// TwinCAT 3 PLC project IDPLC
// ProgramVersion: 3.1.4024.12
// libraries:
//   Tc2_Drive, * (Beckhoff Automation GmbH)
//   Tc2_EtherCAT, * (Beckhoff Automation GmbH)
//   Tc2_Math, * (Beckhoff Automation GmbH)
//   Tc2_MC2, * (Beckhoff Automation GmbH)
//   Tc2_NC, * (Beckhoff Automation GmbH)
//   Tc2_NcDrive, * (Beckhoff Automation GmbH)
//   Tc2_SerialCom, * (Beckhoff Automation GmbH)
//   Tc2_Standard, * (Beckhoff Automation GmbH)
//   Tc2_System, * (Beckhoff Automation GmbH)
//   Tc2_Utilities, * (Beckhoff Automation GmbH)
//   Tc3_Module, * (Beckhoff Automation GmbH)
// project tree:
//   DUTs/ DUT.TcDUT (not stored), DUT_SENSOR_DATAS_1.TcDUT (not stored), DUT_SENSOR_DATAS_8.TcDUT (not stored), DUT_SENSOR_DATAS_2.TcDUT (not stored), DUT_SENSOR_DATAS_3.TcDUT (not stored), DUT_SENSOR_DATAS_4.TcDUT (not stored), DUT_SENSOR_DATAS_5.TcDUT (not stored), DUT_SENSOR_DATAS_6.TcDUT (not stored), DUT_SENSOR_DATAS_7.TcDUT (not stored), Struct_M_Compensation.TcDUT (not stored), Struct_M_lakeshore.TcDUT (not stored), ST_P180.TcDUT (not stored), ST_P182.TcDUT (not stored), ST_P183.TcDUT (not stored), ST_PolarizationParam.TcDUT
//   GVLs/ Global_Variables.TcGVL, Variable_Configuration.TcGVL (not stored)
//   / PlcTask.TcTTO, RecipeManager.TcRMO (not stored), Task_SAFE.TcTTO
//   POUs/0.UserMode/ F_GetSysTime.TcPOU (not stored), UserMode.TcPOU
//   POUs/1.CarrierMode/GapMode/ BCGapMode.TcPOU, GapMode.TcPOU
//   POUs/1.CarrierMode/SingleCarrierMode/ SingleCarrierMode.TcPOU
//   POUs/2.SingleMotorMode/DebugMode/ DebugMode.TcPOU
//   POUs/2.SingleMotorMode/TaperMode/ TaperMode.TcPOU
//   POUs/CommonFB/ExternFB/ FB_LedShow.TcPOU (not stored), FB_PlcEmergencyStop.TcPOU (not stored)
//   POUs/CommonFB/MainFB/ FB_CoupleAxis.TcPOU (not stored), FB_DecoupleAxis.TcPOU (not stored), FB_Move.TcPOU, FB_Power.TcPOU, FB_SetAxisPosition.TcPOU, FB_SetMotorAxisPosition.TcPOU (not stored), FB_SetPhaseLowerMotorAxisPosition.TcPOU, FB_SetPhaseUpperAxisPosition.TcPOU, FB_SetPhaseLowerAxisPosition.TcPOU, FB_SetPhaseUpperMotorAxisPosition.TcPOU, FB_Stop.TcPOU
//   POUs/ MAIN.TcPOU
//   POUs/MainPRG/ FB_CheckCoupleStatus.TcPOU (not stored)
//   POUs/PolarStatusFB/ FB_PolarizationState.TcPOU
//   POUs/RS232/ BackgroundEL.TcPOU (not stored), FB_SerialCom.TcPOU (not stored)
//   POUs/TiltSensor/ FB_Simple_MovingAvg.TcPOU (not stored), SAFE.TcPOU

CONFIGURATION IDPLC
    RESOURCE PLC ON TwinCAT3
        TASK PlcTask(INTERVAL := T#10ms, PRIORITY := 20);
        TASK Task_SAFE(INTERVAL := T#1ms, PRIORITY := 1);
        PROGRAM MAIN WITH PlcTask : MAIN;
        PROGRAM SAFE WITH Task_SAFE : SAFE;
    END_RESOURCE
END_CONFIGURATION

// ---- DUTs/ST_PolarizationParam.TcDUT
TYPE ST_PolarizationParam:
STRUCT
    // HM 水平偏振
    Upper_HM  : LREAL := 0.0;
    Lower_HM  : LREAL := 0.0;

    // VM 垂直偏振 (两种情况)
    Upper_VM1 : LREAL := 42.8;
    Lower_VM1 : LREAL := -42.8;
    Upper_VM2 : LREAL := -42.8;
    Lower_VM2 : LREAL := 42.8;

    // LC 左旋圆偏振
    Upper_LC  : LREAL := 64.2;
    Lower_LC  : LREAL := -21.4;

    // RC 右旋圆偏振
    Upper_RC  : LREAL := -64.2;
    Lower_RC  : LREAL := 21.4;

    // 容差
    Tolerance : LREAL := 2.0;
END_STRUCT
END_TYPE

// ---- GVLs/Global_Variables.TcGVL
//{attribute 'Tc2GvlVarNames'}
VAR_GLOBAL
(*IDControl Ready*)
	IDControlReady:BOOL;
(*Maintenance Mode*)
	MaintenanceMode:BOOL;
	MaintenanceModeLed:BOOL;
(*RecipeDescription*)
	RecipeSavedDate:STRING;
	RecipeDescription:STRING;
(*key Command*)
	btn_Power:BOOL;
	btn_PowerOn: BOOL;
	btn_PowerOff: BOOL;
(*Reset*)
btn_Reset:BOOL;
(*Error Massage*)
	Error:BOOL;
	ErrorID:DINT;
	ErrorDescription:STRING;
(*加载配方参数*)
	LoadRecipeParameters:BOOL;
	loadParametersDone:BOOL;
(*Max Velocity Global*)
	MaxVelocityGlobalVelocity : LREAL;
(*设置光栅bias done *)	
	PositionBiasDone:BOOL;
(*Drive Status*)
	DriveStatus:DINT;//1:Drive Ready;2:Axis is in operation;0:Others
(*回程差*)
	HysteresisError:LREAL;
	HysteresisError_PhaseUpper:LREAL:=0.1;
	HysteresisError_PhaseLower:LREAL:=0.1;
(*光栅漂移误差阈值*)
	LEDriftErrorThreshold:LREAL:=0.001;
	LEDriftErrorThreshold_PhaseUpper:LREAL:=0.001;
	LEDriftErrorThreshold_PhaseLower:LREAL:=0.001;
(*Lag Distance threshold*)
	PosDiff_LeftTopLin: LREAL:=0.5;
	PosDiff_RightTopLin:LREAL:=0.5;
	PosDiff_LeftBottomLin:LREAL:=0.5;
	PosDiff_RightBottomLin:LREAL:=0.5;
	PosDiff_PhaseUpperLin:LREAL:=0.5;
	PosDiff_PhaseLowerLin:LREAL:=0.5;
(*UserMode Threshold*)
	Threshold_UserTopPos: LREAL:=0.5;
	Threshold_UserBottomPos: LREAL:=0.5;
	Threshold_UserLeftPos: LREAL:=0.5;
	Threshold_UserRightPos: LREAL:=0.5;
	Threshold_UserTopVelo: LREAL:=0.5;
	Threshold_UserBottomVelo: LREAL:=0.5;
	Threshold_UserLeftVelo: LREAL:=0.5;
	Threshold_UserRightVelo: LREAL:=0.5;
	//
	Range_UserTaperPos:LREAL:=4.01;
	Range_UserTaperVelo:LREAL:=1.01;
	//Diff_TaperLeftPos:LREAL:=0.01;
	//Diff_TaperLeftVelo:LREAL:=0.2;
	//Diff_TaperRightPos:LREAL:=0.05;
	//Diff_TaperRightVelo:LREAL:=0.5;
	//Taper_BeyondRangePositive:BOOL;
	//Diff_TaperTopPos:LREAL:=0.05;
	//Diff_TaperBottomPos:LREAL:=0.05;
	//Taper_BeyondRangeNegtive:BOOL;
(*BCGap Threshold*)
	Threshold_BCTopPos: LREAL:=0.5;
	Threshold_BCBottomPos: LREAL:=0.5;
	Threshold_BCLeftPos: LREAL:=0.5;
	Threshold_BCRightPos: LREAL:=0.5;
	Threshold_BCTopVelo: LREAL:=0.5;
	Threshold_BCBottomVelo: LREAL:=0.5;
	Threshold_BCLeftVelo: LREAL:=0.5;
	Threshold_BCRightVelo: LREAL:=0.5;
(*DebugMode Threshold*)
	Threshold_TopPos_Debug: LREAL:=4;
	Threshold_BottomPos_Debug: LREAL:=4;
	Threshold_LeftPos_Debug: LREAL:=4;
	Threshold_RightPos_Debug: LREAL:=4;
	//单轴目标位置和当前位置之差，阈值
	Threshold_LeftTopPos_Debug: LREAL:=0.4;	
	Threshold_RightTopPos_Debug: LREAL:=0.4;
	Threshold_LeftBottomPos_Debug: LREAL:=0.4;
	Threshold_RightBottomPos_Debug: LREAL:=0.4;
(*Taper Mode Threshold*)
	Range_TaperPos:LREAL:=5.01;
	Range_TaperVelo:LREAL:=1.01;
	Threshold_TaperLeftPos:LREAL:=0.01;
	Threshold_TaperLeftVelo:LREAL:=0.2;
	Threshold_TaperRightPos:LREAL:=0.05;
	Threshold_TaperRightVelo:LREAL:=0.5;
	Taper_BeyondRangePositive:BOOL;
	Threshold_TaperTopPos:LREAL:=0.05;
	Threshold_TaperBottomPos:LREAL:=0.05;
	Taper_BeyondRangeNegtive:BOOL;
(*SingleCarrierMode threshold*)
	Threshold_TopPos_SingleCarrier: LREAL:=2;
	Threshold_BottomPos_SingleCarrier: LREAL:=2;
	Threshold_LeftPos_SingleCarrier: LREAL:=2;
	Threshold_RightPos_SingleCarrier: LREAL:=2;
	Threshold_TopVelo_SingleCarrier: LREAL:=2;
	Threshold_BottomVelo_SingleCarrier: LREAL:=2;
	Threshold_LeftVelo_SingleCarrier: LREAL:=2;
	Threshold_RightVelo_SingleCarrier: LREAL:=2;
		(*Moving or notmoving*)
	moveDoneAllAxis: BOOL;
	moveStatusLeftTop: BOOL;
	moveStatusRightTop: BOOL;
	moveStatusLeftBottom: BOOL;
	moveStatusRightBottom: BOOL;
	moveStatusPhaseUpper: BOOL;
	moveStatusPhaseLower: BOOL;
	moveStatusAllAxis: BOOL;
	moveStatusAnyAxis: BOOL;
	
	(*Moving or notmoving-Motor*)
	moveDoneAllAxisMotor: BOOL;
	moveStatusLeftTopMotor: BOOL;
	moveStatusRightTopMotor: BOOL;
	moveStatusLeftBottomMotor: BOOL;
	moveStatusRightBottomMotor: BOOL;
	moveStatusPhaseUpperMotor: BOOL;
	moveStatusPhaseLowerMotor: BOOL;
	moveStatusAllAxisMotor: BOOL;
	moveStatusAnyAxisMotor: BOOL;	
	moveStatusGap:BOOL;
(*Compensation Value*)
	M_Compensation:ARRAY[1..18] OF Struct_M_Compensation
:=[
(Encoder:=0,	LeftTop:=0,	RightTop:=0,		LeftBottom:=0,	RightBottom:=0,	InRange:=FALSE),
(Encoder:=5.5,	LeftTop:=5.5,	RightTop:=5.5,	LeftBottom:=5.5,	RightBottom:=5.5,	InRange:=FALSE),
(Encoder:=6.0,	LeftTop:=6.0,	RightTop:=6.0,	LeftBottom:=6.0,	RightBottom:=6.0,	InRange:=FALSE),
(Encoder:=6.5,	LeftTop:=6.5,	RightTop:=6.5,	LeftBottom:=6.5,	RightBottom:=6.5,	InRange:=FALSE),
(Encoder:=7.5,	LeftTop:=7.5,	RightTop:=7.5,	LeftBottom:=7.5,	RightBottom:=7.5,	InRange:=FALSE),
(Encoder:=8.5,	LeftTop:=8.5,	RightTop:=8.5,	LeftBottom:=8.5,	RightBottom:=8.5,	InRange:=FALSE),
(Encoder:=9.5,	LeftTop:=9.5,	RightTop:=9.5,	LeftBottom:=9.5,	RightBottom:=9.5,	InRange:=FALSE),
(Encoder:=10.5,	LeftTop:=10.5,	RightTop:=10.5,	LeftBottom:=10.5,	RightBottom:=10.5,		InRange:=FALSE),
(Encoder:=11.5,	LeftTop:=11.5,	RightTop:=11.5,	LeftBottom:=11.5,	RightBottom:=11.5,		InRange:=FALSE),
(Encoder:=30.0,	LeftTop:=30.0,	RightTop:=30.0,	LeftBottom:=30.0,	RightBottom:=30.0,		InRange:=FALSE),
(Encoder:=100.0,	LeftTop:=100.0,	RightTop:=100.0,	LeftBottom:=100.0,	RightBottom:=100.0,		InRange:=FALSE),
(Encoder:=110.0,	LeftTop:=110.0,	RightTop:=110.0,	LeftBottom:=110.0,	RightBottom:=110.0,		InRange:=FALSE),
(Encoder:=120.0,	LeftTop:=120.0,	RightTop:=120.0,	LeftBottom:=120.0,	RightBottom:=120.0,		InRange:=FALSE),
(Encoder:=130.0,	LeftTop:=130.0,	RightTop:=130.0,	LeftBottom:=130.0,	RightBottom:=130.0,		InRange:=FALSE),
(Encoder:=140.0,	LeftTop:=140.0,	RightTop:=140.0,	LeftBottom:=140.0,	RightBottom:=140.0,		InRange:=FALSE),
(Encoder:=150.0,	LeftTop:=150.0,	RightTop:=150.0,	LeftBottom:=150.0,	RightBottom:=150.0,		InRange:=FALSE),
(Encoder:=160.0,	LeftTop:=160.0,	RightTop:=160.0,	LeftBottom:=160.0,	RightBottom:=160.0,		InRange:=FALSE),
(Encoder:=3000.001,	LeftTop:=3000.001,	RightTop:=3000.001,		LeftBottom:=3000.001,	RightBottom:=3000.001,	InRange:=FALSE)];

(*simulation OR NOT*)
	simulation:BOOL;
(*USELinearEncoeder*)
	USELinearEncoder:BOOL:=TRUE;
(*restartTwinCAT*)
	m_restartTC:BOOL;
(*Plc_EmergencyStop *)
	Plc_EmergencyStop  AT %Q*:BOOL:=TRUE;
(*硬急停*)
	Hardware_EmergencyStop :BOOL:=TRUE;
(*LED*)
	Led_Run  AT %Q*:BOOL;
	Led_Error  AT %Q*:BOOL;
(*LimitSwitch*)
	LS_LeftTop_Far  :BOOL;
	LS_LeftTop_Near  :BOOL;
	LS_RightTop_Far  :BOOL;
	LS_RightTop_Near  :BOOL;
	LS_LeftBottom_Far  :BOOL;
	LS_LeftBottom_Near  :BOOL;
	LS_RightBottom_Far :BOOL;
	LS_RightBottom_Near  :BOOL;
	Unreach_LS_Far:BOOL;
	Unreach_LS_Near:BOOL;
	LS_PhaseUpper_Entrance  :BOOL;
	LS_PhaseUpper_Exit  :BOOL;
	LS_PhaseLower_Entrance :BOOL;
	LS_PhaseLower_Exit  :BOOL;
(*kill switch*)
	KS_LeftTop_Far_Contact1:BOOL;
	KS_LeftTop_Far_Contact2:BOOL;
	KS_RightTop_Far_Contact1:BOOL;
	KS_RightTop_Far_Contact2:BOOL;
	KS_LeftBottom_Far_Contact1:BOOL;
	KS_LeftBottom_Far_Contact2:BOOL;
	KS_RightBottom_Far_Contact1:BOOL;
	KS_RightBottom_Far_Contact2:BOOL;
	KS_PhaseUpper_Exit_Contact1:BOOL;
	KS_PhaseUpper_Exit_Contact2:BOOL;
	KS_PhaseLower_Exit_Contact1:BOOL;
	KS_PhaseLower_Exit_Contact2:BOOL;
	
	KS_LeftTop_Near_Contact1:BOOL;
	KS_LeftTop_Near_Contact2:BOOL;
	KS_RightTop_Near_Contact1:BOOL;
	KS_RightTop_Near_Contact2:BOOL;
	KS_LeftBottom_Near_Contact1:BOOL;
	KS_LeftBottom_Near_Contact2:BOOL;
	KS_RightBottom_Near_Contact1:BOOL;
	KS_RightBottom_Near_Contact2:BOOL;
	KS_PhaseUpper_Entrance_Contact1:BOOL;
	KS_PhaseUpper_Entrance_Contact2:BOOL;
	KS_PhaseLower_Entrance_Contact1:BOOL;
	KS_PhaseLower_Entrance_Contact2:BOOL;
(*E-STOP*)
	KS_CabinetEmergency_contact1:BOOL;
	KS_CabinetEmergency_contact2:BOOL;
	KS_handEmergency1_Contact1:BOOL;
	KS_handEmergency1_Contact2:BOOL;
	KS_handEmergency2_Contact1:BOOL;
	KS_handEmergency2_Contact2:BOOL;
	KS_softEmergency2_Contact:BOOL;
(*AX5805_ErrorAsk*)	
	AX5805_ErrorAsk:BOOL;
(*aixs_ref*)
	LeftTopLin: axis_ref;
	RightTopLin:axis_ref;
	LeftBottomLin:axis_ref;
	RightBottomLin:axis_ref;
	PhaseUpperLin:axis_ref;
	PhaseLowerLin:axis_ref;
(*aixs_ref-motor*)
	LeftTopMotor: axis_ref;
	RightTopMotor:axis_ref;
	LeftBottomMotor:axis_ref;
	RightBottomMotor:axis_ref;
	PhaseUpperMotor:axis_ref;
	PhaseLowerMotor:axis_ref;
(*axis Position*)
	Pos_LeftTopLin: LREAL;
	Pos_RightTopLin:LREAL;
	Pos_LeftBottomLin:LREAL;
	Pos_RightBottomLin:LREAL;
	Pos_PhaseUpperLin:LREAL;
	Pos_PhaseLowerLin:LREAL;
(*axis Position-motor*)
	Pos_LeftTopMotor: LREAL;
	Pos_RightTopMotor:LREAL;
	Pos_LeftBottomMotor:LREAL;
	Pos_RightBottomMotor:LREAL;
	Pos_PhaseUpperMotor:LREAL;
	Pos_PhaseLowerMotor:LREAL;
(*axis Position-Delta*)
	DeltaPos_LeftTop: LREAL;
	DeltaPos_RightTop:LREAL;
	DeltaPos_LeftBottom:LREAL;
	DeltaPos_RightBottom:LREAL;
	DeltaPos_PhaseUpper:LREAL;
	DeltaPos_PhaseLower:LREAL;
(*axis Position-Threshold*)
	ThresholdDeltaPos_LeftTop: LREAL:=0.2;
	ThresholdDeltaPos_RightTop:LREAL:=0.2;
	ThresholdDeltaPos_LeftBottom:LREAL:=0.2;
	ThresholdDeltaPos_RightBottom:LREAL:=0.2;
	ThresholdDeltaPos_PhaseUpper:LREAL:=0.2;
	ThresholdDeltaPos_PhaseLower:LREAL:=0.2;
(*axis Velocity*)
	Velo_LeftTopLin: LREAL;
	Velo_RightTopLin:LREAL;
	Velo_LeftBottomLin:LREAL;
	Velo_RightBottomLin:LREAL;
	Velo_PhaseUpperLin:LREAL;
	Velo_PhaseLowerLin:LREAL;
(*axis Velocity-motor*)
	Velo_LeftTopMotor: LREAL;
	Velo_RightTopMotor:LREAL;
	Velo_LeftBottomMotor:LREAL;
	Velo_RightBottomMotor:LREAL;
	Velo_PhaseUpperMotor:LREAL;
	Velo_PhaseLowerMotor:LREAL;
(*axis Velocity-Delta*)
	DeltaVelo_LeftTop: LREAL;
	DeltaVelo_RightTop:LREAL;
	DeltaVelo_LeftBottom:LREAL;
	DeltaVelo_RightBottom:LREAL;
	DeltaVelo_PhaseUpper:LREAL;
	DeltaVelo_PhaseLower:LREAL;
(*axis Velocity-ThresholdDelta*)
	ThresholdDeltaVelo_LeftTop: LREAL:=0.1;
	ThresholdDeltaVelo_RightTop:LREAL:=0.1;
	ThresholdDeltaVelo_LeftBottom:LREAL:=0.1;
	ThresholdDeltaVelo_RightBottom:LREAL:=0.1;
	ThresholdDeltaVelo_PhaseUpper:LREAL:=0.1;
	ThresholdDeltaVelo_PhaseLower:LREAL:=0.1;
(*axis Torque-motor*)
	Torque_LeftTopLin: LREAL;
	Torque_RightTopLin:LREAL;
	Torque_LeftBottomLin:LREAL;
	Torque_RightBottomLin:LREAL;
	Torque_PhaseUpperLin:LREAL;
	Torque_PhaseLowerLin:LREAL;
(*axis Torque-motor*)
	Torque_LeftTopMotor: LREAL;
	Torque_RightTopMotor:LREAL;
	Torque_LeftBottomMotor:LREAL;
	Torque_RightBottomMotor:LREAL;
	Torque_PhaseUpperMotor:LREAL;
	Torque_PhaseLowerMotor:LREAL;
(*axis Torque-Delta*)
	DeltaTorque_LeftTop: LREAL;
	DeltaTorque_RightTop:LREAL;
	DeltaTorque_LeftBottom:LREAL;
	DeltaTorque_RightBottom:LREAL;
	DeltaTorque_PhaseUpper:LREAL;
	DeltaTorque_PhaseLower:LREAL;
(*Lag Distance*)
	PosDiff_LeftTopLin_actual: LREAL;
	PosDiff_RightTopLin_actual:LREAL;
	PosDiff_LeftBottomLin_actual:LREAL;
	PosDiff_RightBottomLin_actual:LREAL;
	PosDiff_PhaseUpperLin_actual:LREAL;
	PosDiff_PhaseLowerLin_actual:LREAL;
(*Lag Distance-Motor*)
	PosDiff_LeftTopMotor_actual: LREAL;
	PosDiff_RightTopMotor_actual:LREAL;
	PosDiff_LeftBottomMotor_actual:LREAL;
	PosDiff_RightBottomMotor_actual:LREAL;
	PosDiff_PhaseUpperMotor_actual:LREAL;
	PosDiff_PhaseLowerMotor_actual:LREAL;
(*Delta LagDistance*)
	DeltaPosDiff_LeftTop_actual: LREAL;
	DeltaPosDiff_RightTop_actual:LREAL;
	DeltaPosDiff_LeftBottom_actual:LREAL;
	DeltaPosDiff_RightBottom_actual:LREAL;
	DeltaPosDiff_PhaseUpper_actual:LREAL;
	DeltaPosDiff_PhaseLower_actual:LREAL;
(********************Gap Mode*************************)
(**)
	GapPositionActual:LREAL;
	GapVelocityActual:LREAL;
	GapMoveIndicator:DINT:=0;
	(*1=OPEN;0=NOTMOVE;-1=CLOSE*)
(******************Taper Mode**************************)
(*Taper*)
	TaperPositionActual:LREAL;
	TaperVelocityActual:LREAL;
	TaperMoveIndicator:DINT:=0;
	(*1=OPEN;0=NOTMOVE;-1=CLOSE*)
(*****************singleCarrier Mode*******************************)
(**)
	TopPositionActual:LREAL;
	TopVelocityActual:LREAL;
	BottomPositionActual:LREAL;
	BottomVelocityActual:LREAL;
	TopMoveIndicator:DINT:=0;
	(*1=OPEN;0=NOTMOVE;-1=CLOSE*)
	BottomMoveIndicator:DINT:=0;
	(*1=OPEN;0=NOTMOVE;-1=CLOSE*)
(******************DebugMode & BCGapMode*****************************)
	LeftTopLinMoveIndicator:DINT:=0;
	(*1=OPEN;0=NOTMOVE;-1=CLOSE*)
	LeftBottomLinMoveIndicator:DINT:=0;
	(*1=OPEN;0=NOTMOVE;-1=CLOSE*)
	RightTopLinMoveIndicator:DINT:=0;
	(*1=OPEN;0=NOTMOVE;-1=CLOSE*)
	RightBottomLinMoveIndicator:DINT:=0;
	(*1=OPEN;0=NOTMOVE;-1=CLOSE*)
(******************Gap&SingleCarrier***********************************)
	Diff_TopPos_actual: LREAL;
	Diff_BottomPos_actual: LREAL;
	Diff_LeftPos_actual: LREAL;
	Diff_RightPos_actual: LREAL;
	Diff_TopVelo_actual:  LREAL;
	Diff_BottomVelo_actual: LREAL;
	Diff_LeftVelo_actual: LREAL;
	Diff_RightVelo_actual:  LREAL;

(******************BCGap Mode***********************************)
	Diff_BCTopPos_actual: LREAL;
	Diff_BCBottomPos_actual: LREAL;
	Diff_BCLeftPos_actual: LREAL;
	Diff_BCRightPos_actual: LREAL;
	Diff_BCTopVelo_actual:  LREAL;
	Diff_BCBottomVelo_actual: LREAL;
	Diff_BCLeftVelo_actual: LREAL;
	Diff_BCRightVelo_actual:  LREAL;
(******************UserMode*********************)
	Diff_UserTopPos_actual: LREAL;
	Diff_UserBottomPos_actual: LREAL;
	Diff_UserLeftPos_actual: LREAL;
	Diff_UserRightPos_actual: LREAL;
	Diff_UserTopVelo_actual:  LREAL;
	Diff_UserBottomVelo_actual: LREAL;
	Diff_UserLeftVelo_actual: LREAL;
	Diff_UserRightVelo_actual:  LREAL;
	TaperFunctionSolidOn:BOOL;//该ID是否有taper需求，taper总开关，只在参数表生效
	TaperOrNot:BOOL;
	UserTaperPositionActual:LREAL;
	UserTaperVelocityActual:LREAL;
(***********************Power status and couple statatus***********************)
	st_Power:BOOL;
	st_Couple:DINT;
(************************FB***********************)
	FB_Power:FB_Power;
	FB_PlcEmergencyStop: FB_PlcEmergencyStop;
	FB_CheckCoupleStatus:FB_CheckCoupleStatus;
	FB_Move:FB_Move;
	FB_Stop:FB_Stop;
	FB_DecoupleAxis:FB_DecoupleAxis;
	FB_CoupleAxis: FB_CoupleAxis;
	FB_Move_PhaseUpper:FB_Move;
	FB_Stop_PhaseUpper:FB_Stop;
	FB_Move_PhaseLower:FB_Move;
	FB_Stop_PhaseLower:FB_Stop;
(********************²¹³¥GapÄ£Ê½£¬µ¥Öá²¹³¥Êý¾Ý************************)
	(*ÊÇ·ñ²¹³¥*)
	USE_SingleAxis_Compensation:BOOL:=TRUE;
	Mdut:ARRAY[1..2] OF DUT:=
	[(Encoder:=2.0,	LeftTop:=2.3000),
	(Encoder:=2.0,	LeftTop:=2.3000)];


	M_CompensationNumber:INT;
	M_DisplayNumber:INT;
	(*Conpensation Position Target*)
	LeftTopLinPositionNew:LREAL;
	LeftBottomLinPositionNew:LREAL;
	RightTopLinPositionNew:LREAL;
	RightBottomLinPositionNew:LREAL;
	(*考虑到回程差后，运动到临时位置*)
	LeftTopLinPositionNew_temporary :LREAL;
	LeftBottomLinPositionNew_temporary:LREAL;
	RightTopLinPositionNew_temporary:LREAL;
	RightBottomLinPositionNew_temporary:LREAL;
	(*Display Position*)
	LeftTopLinPositionDisplay:LREAL;
	LeftBottomLinPositionDisplay:LREAL;
	RightTopLinPositionDisplay:LREAL;
	RightBottomLinPositionDisplay:LREAL;
	(*Display Velocity*)
	LeftTopLinVelocityDisplay:LREAL;
	LeftBottomLinVelocityDisplay:LREAL;
	RightTopLinVelocityDisplay:LREAL;
	RightBottomLinVelocityDisplay:LREAL;
	(*temperature sensors*)
	thermocouple AT %I*:ARRAY[1..12]OF  DINT;
	shieldPt100  AT %I*:ARRAY[1..12]OF INT;
	thermocouple_Celsius:ARRAY[1..12]OF  LREAL;
	shieldPt100_Celsius  :ARRAY[1..12]OF LREAL;
	huoer_Celsius AT %I* :ARRAY[1..3]OF INT;
	(**)
	lakeshorePt100  AT %I*:ARRAY[1..12]OF INT;(*16*×èÖµ*)
	lakeshorePt100_Resistance :ARRAY[1..12]OF LREAL;(*ÉãÊÏÎÂ¶È*)
	lakeshorePt100_Celsius  :ARRAY[1..12]OF LREAL;(*ÉãÊÏÎÂ¶È*)
	temperatureCompensationValue:LREAL:=6;
	testSensors  AT %I*:ARRAY[1..4]OF INT;

(******RS232************)
	RxBufferEL			: ComBuffer;	(* Receive data buffer; used with all receive function blocks *)
	TxBufferEL			: ComBuffer;	(* Transmit data buffer; used with all receive function blocks *)
(*input protection*)
	//
	min_UserGapPositionNew:LREAL:=10;
	max_UserGapPositionNew:LREAL:=200;
	inRange_UserGapPositionNew:BOOL;
	//LE protection position
	min_UserLEProtectionGapPosition:LREAL;
	min_ThresholdGapSoft2LEProtection:LREAL;
	max_UserLEProtectionGapPosition:LREAL;
	max_ThresholdGapSoft2LEProtection:LREAL;
	//
	min_UserGapVelocityNew:LREAL:=0;
	max_UserGapVelocityNew:LREAL:=2;
	inRange_UserGapVelocityNew:BOOL;
	//
	min_UserPhaseUpperPositionNew:LREAL:=-10;
	max_UserPhaseUpperPositionNew:LREAL:=10;
	inRange_UserPhaseUpperPositionNew:BOOL;
	//LE protection position
	min_UserLEProtectionPhaseUpperPosition:LREAL;
	max_UserLEProtectionPhaseUpperPosition:LREAL;
	min_ThresholdPhaseUpperSoft2LEProtection:LREAL;
	max_ThresholdPhaseUpperSoft2LEProtection:LREAL;
	//
	min_UserPhaseUpperVelocityNew:LREAL:=0;
	max_UserPhaseUpperVelocityNew:LREAL:=1;
	inRange_UserPhaseUpperVelocityNew:BOOL;
	//
	min_UserPhaseLowerPositionNew:LREAL:=-10;
	max_UserPhaseLowerPositionNew:LREAL:=10;
	inRange_UserPhaseLowerPositionNew:BOOL;
	//LE protection position
	min_UserLEProtectionPhaseLowerPosition:LREAL;
	max_UserLEProtectionPhaseLowerPosition:LREAL;
	min_ThresholdPhaseLowerSoft2LEProtection:LREAL;
	max_ThresholdPhaseLowerSoft2LEProtection:LREAL;
	//
	min_UserPhaseLowerVelocityNew:LREAL:=0;
	max_UserPhaseLowerVelocityNew:LREAL:=1;
	inRange_UserPhaseLowerVelocityNew:BOOL;
	//
	min_UserTaperPositionNew: LREAL:=0;;
	max_UserTaperPositionNew: LREAL:=0;
	inRange_UserTaperPositionNew: BOOL;
	//
	min_UserTaperVelocityNew: LREAL:=0;
	max_UserTaperVelocityNew: LREAL:=0;
	inRange_UserTaperVelocityNew: BOOL;
	
		(*add Beamline taper 模式，入口和出口电机都运动，保持中心gap不变*)
	//3种模式划分：
	NormalGapMode:BOOL;
	IDTaperMode:BOOL;
	BLTaperMode:BOOL;
	
END_VAR

// ---- POUs/MAIN.TcPOU
PROGRAM MAIN
VAR
	pbGapMode: BOOL:=FALSE;
	pbTaperMode: BOOL:=FALSE;
	pbSingleCarrierMode: BOOL:=FALSE;
	pbDebugMode:BOOL:=FALSE;
	pbBCGapMode:BOOL:=FALSE;
	fb_led_Show: FB_LedShow;
	btn_reset: BOOL;
	CPMU_PLC_Reset: PLC_Reset;
	d_state: DINT;
	CPMU_PLC_Start: PLC_Start;
	powerStatus:BOOL;

(*TwinSAFE*)
	Safe_run AT%Q*:BOOL;
	Err_Ack AT %Q*:BOOL;
	Estop_RunAndRestart AT %Q*:BOOL;
	AX5805_Error_Ack AT %Q*:BOOL;
	Led_Run  AT %Q*:BOOL;
	Led_Error  AT %Q*:BOOL;

	FB_ERROR AT%I*:BOOL;
	COM_ERROR AT%I*:BOOL;
	//OUT_ERROR AT%I*:BOOL;
	Estop_Out AT%I*:BOOL;

	SafeStatus:INT;
	SafePLCRunOK: BOOL;
	fb_ton: TON;
	fb_ton2: TON;
	fb_ton3: TON;
	fb_ton1: TON;
	fb_ton0: TON;
(*IO*)
	el1808_D1  AT%I* :ARRAY[1..12] OF BOOL;
	el1808_D2  AT%I* :ARRAY[1..4] OF BOOL;
	el1008 AT%I*:BOOL;
	EStopTrig:BOOL;
(*setAxisPosition*)
	SetAxisPosState: INT;
	FB_Set_AxisPosition:FB_SetAxisPosition;
	fb_ton4: TON;
	fb_ton5: TON;
	fb_ton6: TON;
	SetAxisPositionDone: BOOL;
	//
	SetPhaseUpperAxisPosState: INT;
	FB_Set_PhaseUpperAxisPosition:FB_SetPhaseUpperAxisPosition;
	fb_ton7: TON;
	fb_ton8: TON;
	fb_ton9: TON;
	SetPhaseUpperAxisPositionDone: BOOL;
	//
	SetPhaseLowerAxisPosState: INT;
	FB_Set_PhaseLowerAxisPosition:FB_SetPhaseLowerAxisPosition;
	fb_ton10: TON;
	fb_ton11: TON;
	fb_ton12: TON;
	SetPhaseLowerAxisPositionDone: BOOL;
	i: INT;
	j: INT;

(****RS232***)
	fbEL6001	: FB_SerialCom;
	moveDoneLeftTop: BOOL;
	moveDoneRightTop: BOOL;
	moveDoneLeftBottom: BOOL;
	moveDoneRightBottom: BOOL;

(*Torque*)
	Torque_LT AT%I*:INT;
	Torque_RT AT%I*:INT;
	Torque_LB AT%I*:INT;
	Torque_RB AT%I*:INT;
	Torque_PU AT%I*:INT;
	Torque_PL AT%I*:INT;
(**)
	btn_setAxisPosition: BOOL;
	ValueSet_LeftTop:LREAL;
	ValueSet_RightTop:LREAL;
	ValueSet_LeftBottom:LREAL;
	ValueSet_RightBottom:LREAL;
	btn_setPhaseUpperAxisPosition: BOOL;
	PhaseUpperSetValue: LREAL;
	btn_setPhaseLowerAxisPosition: BOOL;
	PhaseLowerSetValue: LREAL;
(**)
	RestartTC: TC_Restart;
	
(*recipe*)
	RecipeINT:INT;
	RecipeBOOL:BOOL;
	RecipeManCommands: RecipeManCommands;
	SaveParameter : BOOL;  //保存文件
	LoadParameter : BOOL;  //读取文件
	Save_R_TRIG   : R_TRIG;
	Read_R_TRIG   : R_TRIG;
	loadparameterStatus: INT;
	RecipeBOOL2:BOOL;
	ReturnDwordLoad: DWORD;
	InsertionDeviceName:STRING;
(*UserMode*)
	pbUserMode: BOOL:=TRUE;
	EL1904 AT%I* :ARRAY[1..32] OF BOOL;
	setAxisPositionEnable: BOOL;
	setPhaseUpperAxisPositionEnable: BOOL;
	setPhaseLowerAxisPositionEnable: BOOL;
	state_loadParameters: INT;
	state_setLEPosBias: INT;
	//
	PositionBiasSet:BOOL;
	MC_SetLEPosBias_LeftTop:MC_WriteParameter;
	MC_SetLEPosBias_RightTop:MC_WriteParameter;
	MC_SetLEPosBias_LeftBottom:MC_WriteParameter;
	MC_SetLEPosBias_RightBottom:MC_WriteParameter;
	MC_SetLEPosBias_PhaseUpper:MC_WriteParameter;
	MC_SetLEPosBias_PhaseLower:MC_WriteParameter;
	PositionBias_LeftTop: LREAL:=10.1;
	PositionBias_RightTop: LREAL:=10.2;
	PositionBias_LeftBottom: LREAL:=10.3;
	PositionBias_RightBottom: LREAL:=10.4;
	PositionBias_PhaseUpper: LREAL:=10.3;
	PositionBias_PhaseLower: LREAL:=10.4;
	
	LoadLEPB_R_TRIG: R_TRIG;
	PositionBiasTON: TON;
	
	//
	OPC_TEST_Bi:BOOL:=TRUE; (*~ (OPC:1:available for OPC Clients) *)
	OPC_TEST_Bi2:BOOL;(*~ (OPC:1:available for OPC Clients) *)
	//
	HasTemperatureSensorOrNot:BOOL;//Only IVU or CPMU
	(*Sensor Reading*)
	Sensor_Reading_1 AT %I*:ARRAY[0..3] OF BYTE;
	Sensor_Reading_2 AT %I*:ARRAY[0..3] OF BYTE;
	Sensor_Reading_3 AT %I*:ARRAY[0..3] OF BYTE;
	Sensor_Reading_4 AT %I*:ARRAY[0..3] OF BYTE;
	Sensor_Reading_5 AT %I*:ARRAY[0..3] OF BYTE;
	Sensor_Reading_6 AT %I*:ARRAY[0..3] OF BYTE;
	Sensor_Reading_7 AT %I*:ARRAY[0..3] OF BYTE;
	Sensor_Reading_8 AT %I*:ARRAY[0..3] OF BYTE;
	Sensor_Reading_DpState AT %I*:USINT;
	Sensor_Reading_ExtDiagFlag AT %I*:BOOL;
	TemperatureSensors_1:LREAL;
	TemperatureSensors_2:LREAL;
	TemperatureSensors_3:LREAL;
	TemperatureSensors_4:LREAL;
	TemperatureSensors_5:LREAL;
	TemperatureSensors_6:LREAL;
	TemperatureSensors_7:LREAL;
	TemperatureSensors_8:LREAL;
	dut_sensor_datas_1:DUT_SENSOR_DATAS_1;
	dut_sensor_datas_2:DUT_SENSOR_DATAS_2;
	dut_sensor_datas_3:DUT_SENSOR_DATAS_3;
	dut_sensor_datas_4:DUT_SENSOR_DATAS_4;
	dut_sensor_datas_5:DUT_SENSOR_DATAS_5;
	dut_sensor_datas_6:DUT_SENSOR_DATAS_6;
	dut_sensor_datas_7:DUT_SENSOR_DATAS_7;
	dut_sensor_datas_8:DUT_SENSOR_DATAS_8;
	//
	temperature_gradient_2_To_1:LREAL;
	temperature_gradient_3_To_2:LREAL;
	temperature_gradient_5_To_4:LREAL;
	temperature_gradient_6_To_5:LREAL;
	temperature_gradient_max:LREAL;
	//
	temperature_average:LREAL;
	A_SetLinearEncoderPositionBias_Enable: BOOL;
	
		//
	temperatureStatus:INT;//0：有传感器度数错误；1:常温；2:低温；3:常温和低温中间态
	CryogenicTemperatureThreshold:LREAL:=80;//80K以下归划分为低温
	RoomTemperatureThreshold:LREAL:=293;//293K以上划分为常温
	//CPMU cryogenix ON/FF
	CryogenicCompensationOn:BOOL;
	CryogenicCompensationConditionsReady:BOOL;
	CryogenicCompensation_LeftTop:LREAL;
	CryogenicCompensation_RightTop:LREAL;
	CryogenicCompensation_LeftBottom:LREAL;
	CryogenicCompensation_RightBottom:LREAL;
	CryogenicCompensationDone: BOOL;
	
	(**)
	bDriveDiagMessageAndNumber  : BOOL;
	m_GetDriveStatusState:INT;
	GetDriveStatusStateDone:BOOL;
	GetDriveStatusStateError:BOOL;
	//	
	fb_SoEReadDiagMessage_LeftTop: FB_SoEReadDiagMessage;
	fb_SoEReadDiagMessage_RightTop: FB_SoEReadDiagMessage;
	fb_SoEReadDiagMessage_LeftBottom: FB_SoEReadDiagMessage;
	fb_SoEReadDiagMessage_RightBottom: FB_SoEReadDiagMessage;
	fb_SoEReadDiagMessage_PhaseUpper: FB_SoEReadDiagMessage;
	fb_SoEReadDiagMessage_PhaseLower: FB_SoEReadDiagMessage;
	DriveDiagMessage_LeftTop:STRING;
	DriveDiagMessage_RightTop:STRING;
	DriveDiagMessage_LeftBottom:STRING;
	DriveDiagMessage_RightBottom:STRING;
	DriveDiagMessage_PhaseUpper:STRING;
	DriveDiagMessage_PhaseLower:STRING;
	//
	FB_SoEReadDiagNumber_LeftTop: FB_SoEReadDiagNumber;
	FB_SoEReadDiagNumber_RightTop: FB_SoEReadDiagNumber;
	FB_SoEReadDiagNumber_LeftBottom: FB_SoEReadDiagNumber;
	FB_SoEReadDiagNumber_RightBottom: FB_SoEReadDiagNumber;
	FB_SoEReadDiagNumber_PhaseUpper: FB_SoEReadDiagNumber;
	FB_SoEReadDiagNumber_PhaseLower: FB_SoEReadDiagNumber;
	DriveDiagNumber_LeftTop:UDINT;
	DriveDiagNumber_RightTop:UDINT;
	DriveDiagNumber_LeftBottom:UDINT;
	DriveDiagNumber_RightBottom:UDINT;
	DriveDiagNumber_PhaseUpper:UDINT;
	DriveDiagNumber_PhaseLower:UDINT;
	bReloadDriveDiagMessageAndNumber: BOOL;
	
	(*load IOC*)
	bExe_load_Prog: BOOL;
	NT_StartProcess_Load: NT_StartProcess;
	Exe_load_step: UINT;
	R_TRIG_ExeLoad: R_TRIG;
	Exe_Load_Done:BOOL;
	(*kill IOC*)
	bExe_Kill_Prog: BOOL;
	NT_StartProcess_Kill: NT_StartProcess;
	Exe_kill_step: UINT;
	R_TRIG_Exekill: R_TRIG;
	Exe_Kill_Done:BOOL;
	LoadOpcIocTON:TON;
	
	GetDriveStatusTON:TON;
	
	//
	//more parameters get:gear;feedback2 direction 
	//
	//GetMoreDriveStatus_FunctionON:BOOL:=TRUE;
	GetDriveStatusTON2: TON;
	//GearNumerator,st182
	st_p182_LeftTop:ST_P182;
	FB_SoERead_GearNumerator_LeftTop: FB_SoERead;
	st_p182_RightTop:ST_P182;
	FB_SoERead_GearNumerator_RightTop: FB_SoERead;
	st_p182_LeftBottom:ST_P182;
	FB_SoERead_GearNumerator_LeftBottom: FB_SoERead;
	st_p182_RightBottom:ST_P182;
	FB_SoERead_GearNumerator_RightBottom: FB_SoERead;
	st_p182_PhaseUpper:ST_P182;
	FB_SoERead_GearNumerator_PhaseUpper: FB_SoERead;
	st_p182_PhaseLower:ST_P182;
	FB_SoERead_GearNumerator_PhaseLower: FB_SoERead;
	GearNumeratorGet_LeftTop:UDINT;
	GearNumeratorGet_RightTop:UDINT;
	GearNumeratorGet_LeftBottom:UDINT;
	GearNumeratorGet_RightBottom:UDINT;
	GearNumeratorGet_PhaseUpper:UDINT;
	GearNumeratorGet_PhaseLower:UDINT;
	GearNumeratorConfigured_LeftTop:UDINT;
	GearNumeratorConfigured_RightTop:UDINT;
	GearNumeratorConfigured_LeftBottom:UDINT;
	GearNumeratorConfigured_RightBottom:UDINT;
	GearNumeratorConfigured_PhaseUpper:UDINT;
	GearNumeratorConfigured_PhaseLower:UDINT;
	//GearDenominator,st183
	st_p183_LeftTop:ST_P183;
	FB_SoERead_GearDenominator_LeftTop: FB_SoERead;
	st_p183_RightTop:ST_P183;
	FB_SoERead_GearDenominator_RightTop: FB_SoERead;
	st_p183_LeftBottom:ST_P183;
	FB_SoERead_GearDenominator_LeftBottom: FB_SoERead;
	st_p183_RightBottom:ST_P183;
	FB_SoERead_GearDenominator_RightBottom: FB_SoERead;
	st_p183_PhaseUpper:ST_P183;
	FB_SoERead_GearDenominator_PhaseUpper: FB_SoERead;
	st_p183_PhaseLower:ST_P183;
	FB_SoERead_GearDenominator_PhaseLower: FB_SoERead;
	GearDenominatorGet_LeftTop:UDINT;
	GearDenominatorGet_RightTop:UDINT;
	GearDenominatorGet_LeftBottom:UDINT;
	GearDenominatorGet_RightBottom:UDINT;
	GearDenominatorGet_PhaseUpper:UDINT;
	GearDenominatorGet_PhaseLower:UDINT;
	GearDenominatorConfigured_LeftTop:UDINT;
	GearDenominatorConfigured_RightTop:UDINT;
	GearDenominatorConfigured_LeftBottom:UDINT;
	GearDenominatorConfigured_RightBottom:UDINT;
	GearDenominatorConfigured_PhaseUpper:UDINT;
	GearDenominatorConfigured_PhaseLower:UDINT;
	//Feedback2direction,st180
	st_p180_LeftTop:ST_P180;
	FB_SoERead_Feedback2direction_LeftTop: FB_SoERead;
	st_p180_RightTop:ST_P180;
	FB_SoERead_Feedback2direction_RightTop: FB_SoERead;
	st_p180_LeftBottom:ST_P180;
	FB_SoERead_Feedback2direction_LeftBottom: FB_SoERead;
	st_p180_RightBottom:ST_P180;
	FB_SoERead_Feedback2direction_RightBottom: FB_SoERead;
	st_p180_PhaseUpper:ST_P180;
	FB_SoERead_Feedback2direction_PhaseUpper: FB_SoERead;
	st_p180_PhaseLower:ST_P180;
	FB_SoERead_Feedback2direction_PhaseLower: FB_SoERead;
	Feedback2directionGet_LeftTop:UINT;
	Feedback2directionGet_RightTop:UINT;
	Feedback2directionGet_LeftBottom:UINT;
	Feedback2directionGet_RightBottom:UINT;
	Feedback2directionGet_PhaseUpper:UINT;
	Feedback2directionGet_PhaseLower:UINT;
	Feedback2directionConfigured_LeftTop:UINT;
	Feedback2directionConfigured_RightTop:UINT;
	Feedback2directionConfigured_LeftBottom:UINT;
	Feedback2directionConfigured_RightBottom:UINT;
	Feedback2directionConfigured_PhaseUpper:UINT;
	Feedback2directionConfigured_PhaseLower:UINT;
	
	//RestartDrivers
		(*重启驱动器*)
	btn_RestartDriversAll:BOOL;
	btn_RestartDriver1:BOOL;
	btn_RestartDriver2:BOOL;
	btn_RestartDriver3:BOOL;
	btn_RestartDriver4:BOOL;
	btn_RestartDriver5:BOOL;
	btn_RestartDriver6:BOOL;
	btn_RestartDriver7:BOOL;
	btn_RestartDriver8:BOOL;
	Relay_EL2624 AT %Q*:ARRAY[0..7]OF  BOOL;
	RestartDriver_RTRIG:R_TRIG;
	RestartDriver_TON:TON;
	RestartDriver_Triggered:BOOL;
	RestartDriver_State:DINT;
	RestartDriver_Done:BOOL;
	//
	
	//
	//	LEHeartBeatMonitorFunction
	//
	LEHeartBeatMonitorFunctionOn: BOOL;
	LEHeartBeatFirstScan:BOOL;
	LEHeartBeatDeadZone : LREAL := 0; 
	LEHeartBeatAlarmTime : TIME := T#0.1S;
	
    //Pos_LeftTopLin_Last : LREAL; 
	Velo_LeftTopLin_Last : LREAL; 
	Pos_LeftTopMotor_Initial : LREAL; 
    StableTimer_LeftTopLin : TON; 
    StableTime_LeftTopLin : TIME; 
    DeltaVelo_LeftTopLin : LREAL; 
	IsInitialPositionSet_LeftTop: BOOL;
	MotorPosChange_LeftTop: LREAL;
	Threshold_LeftTopMotorPos:LREAL:=0.1;
	Threshold_LeftTopMotorVelo:LREAL:=0.2;
	Alarm_LeftTopLin:BOOL;
	Alarm_LeftTopMotorPos:BOOL;
	Alarm_LeftTopMotorVelo:BOOL;
	
	
	//Pos_RightTopLin_Last : LREAL; 
	Velo_RightTopLin_Last : LREAL; 
	Pos_RightTopMotor_Initial : LREAL; 
    StableTimer_RightTopLin : TON; 
    StableTime_RightTopLin : TIME; 
    DeltaVelo_RightTopLin : LREAL; 
	IsInitialPositionSet_RightTop: BOOL;
	MotorPosChange_RightTop: LREAL; 
	Threshold_RightTopMotorPos:LREAL:=0.1;
	Threshold_RightTopMotorVelo:LREAL:=0.2;
	Alarm_RightTopLin:BOOL;
	Alarm_RightTopMotorPos:BOOL;
	Alarm_RightTopMotorVelo:BOOL;
	
		
    //Pos_LeftBottomLin_Last : LREAL; 
	Velo_LeftBottomLin_Last : LREAL; 
	Pos_LeftBottomMotor_Initial : LREAL; 
    StableTimer_LeftBottomLin : TON; 
    StableTime_LeftBottomLin : TIME; 
    DeltaVelo_LeftBottomLin : LREAL; 
	IsInitialPositionSet_LeftBottom: BOOL;
	MotorPosChange_LeftBottom: LREAL; 
	Threshold_LeftBottomMotorPos:LREAL:=0.1;
	Threshold_LeftBottomMotorVelo:LREAL:=0.2;
	Alarm_LeftBottomLin:BOOL;
	Alarm_LeftBottomMotorPos:BOOL;
	Alarm_LeftBottomMotorVelo:BOOL;
	
	//Pos_RightBottomLin_Last : LREAL; 
	Velo_RightBottomLin_Last : LREAL; 
	Pos_RightBottomMotor_Initial : LREAL; 
    StableTimer_RightBottomLin : TON; 
    StableTime_RightBottomLin : TIME; 
    DeltaVelo_RightBottomLin : LREAL; 
	IsInitialPositionSet_RightBottom: BOOL;
	MotorPosChange_RightBottom: LREAL; 
	Threshold_RightBottomMotorPos:LREAL:=0.1;
	Threshold_RightBottomMotorVelo:LREAL:=0.2;
	Alarm_RightBottomLin:BOOL;
	Alarm_RightBottomMotorPos:BOOL;
	Alarm_RightBottomMotorVelo:BOOL;
	
	//Pos_PhaseUpperLin_Last : LREAL; 
	Velo_PhaseUpperLin_Last : LREAL; 
	Pos_PhaseUpperMotor_Initial : LREAL; 
    StableTimer_PhaseUpperLin : TON; 
    StableTime_PhaseUpperLin : TIME; 
    DeltaVelo_PhaseUpperLin : LREAL; 
	IsInitialPositionSet_PhaseUpper: BOOL;
	MotorPosChange_PhaseUpper: LREAL; 
	Threshold_PhaseUpperMotorPos:LREAL:=0.1;
	Threshold_PhaseUpperMotorVelo:LREAL:=0.2;
	Alarm_PhaseUpperLin:BOOL;
	Alarm_PhaseUpperMotorPos:BOOL;
	Alarm_PhaseUpperMotorVelo:BOOL;
	
	//Pos_PhaseLowerLin_Last : LREAL; 
	Velo_PhaseLowerLin_Last : LREAL; 
	Pos_PhaseLowerMotor_Initial : LREAL; 
    StableTimer_PhaseLowerLin : TON; 
    StableTime_PhaseLowerLin : TIME; 
    DeltaVelo_PhaseLowerLin : LREAL; 
	IsInitialPositionSet_PhaseLower: BOOL;
	MotorPosChange_PhaseLower: LREAL; 
	Threshold_PhaseLowerMotorPos:LREAL:=0.1;
	Threshold_PhaseLowerMotorVelo:LREAL:=0.2;
	Alarm_PhaseLowerLin:BOOL;
	Alarm_PhaseLowerMotorPos:BOOL;
	Alarm_PhaseLowerMotorVelo:BOOL;
	
	(*setAxisPosition*)
	SetMotorAxisPosState: INT;
	FB_Set_MotorAxisPosition:FB_SetMotorAxisPosition;
	fb_ton4_2: TON;
	fb_ton5_2: TON;
	SetMotorAxisPositionDone: BOOL;
	btn_SetMotorAxisPosition: BOOL;	
	(*setAxisPosition-PhaseUpper*)
	SetPhaseUpperMotorAxisPosState: INT;
	FB_Set_PhaseUpperMotorAxisPosition:FB_SetPhaseUpperMotorAxisPosition;
	fb_ton7_2: TON;
	SetPhaseUpperMotorAxisPositionDone: BOOL;
	btn_SetPhaseUpperMotorAxisPosition: BOOL;
	(*setAxisPosition-PhaseLower*)
	SetPhaseLowerMotorAxisPosState: INT;
	FB_Set_PhaseLowerMotorAxisPosition:FB_SetPhaseLowerMotorAxisPosition;
	fb_ton8_2: TON;
	SetPhaseLowerMotorAxisPositionDone: BOOL;
	btn_SetPhaseLowerMotorAxisPosition: BOOL;
	
	
	MonitorMotorAndLEFunctionOn:BOOL:=TRUE;
	
		(*GetMotorTempture*)
	MotorTemperature AT %I*:ARRAY[0..5] OF UINT;
	MotorTemperature_LeftTop:LREAL;
	MotorTemperature_RightTop:LREAL;
	MotorTemperature_LeftBottom:LREAL;
	MotorTemperature_RightBottom:LREAL;
	MotorTemperature_PhaseUpper:LREAL;
	MotorTemperature_PhaseLower:LREAL;

	fbPolar    : FB_PolarizationState;
    stPolarizationParam   : ST_PolarizationParam;
END_VAR

(*MaintenanceMode*)
IF MaintenanceMode THEN
	MaintenanceModeLed:=TRUE;
	RETURN;
ELSE
	MaintenanceModeLed:=FALSE;	
END_IF
(*加载Ricipe参数*)
A_InitRecipeParameters();
(*Restart TwinCAT*)
IF Global_Variables.m_restartTC THEN
(*首先关闭opcIocShell.exe*)	
	bExe_Kill_Prog:=TRUE;
	A_KillOpcIocShellExe();
(*重启TC*)
	IF Exe_Kill_Done THEN
		A_RestartTC();
	END_IF
END_IF
(*******InitAxisParameters*******)
A_InitAxisParameters();
(*******¼à²âÏÞÎ»¿ª¹Ø×´Ì¬£¬·½Ïò¿ØÖÆ&½ô¼±Çé¿öÏÂEStop*******)
A_CheckLimitSwitch();
(*Check Kill Switch*)
A_CheckKillSwitch();
(*******PosDiff¼à¿Ø*******)
A_PosDiffDetectiion();
(*******³õÊ¼»¯SafePlc*******)
IF NOT simulation THEN
A_SafePlcStartInit();
END_IF
(************SetAxisPosition-GAP*********************)
IF  NOT USELinearEncoder AND setAxisPositionEnable AND btn_setAxisPosition THEN
		FB_Set_AxisPosition.ValueSet_LeftTop:=ValueSet_LeftTop;
		FB_Set_AxisPosition.ValueSet_RightTop:=ValueSet_RightTop;
		FB_Set_AxisPosition.ValueSet_LeftBottom:=ValueSet_LeftBottom;
		FB_Set_AxisPosition.ValueSet_RightBottom:=ValueSet_RightBottom;
		A_SetAxisPosition();
END_IF
(************SetAxisPosition-GAP*********************)
IF  NOT USELinearEncoder AND setPhaseUpperAxisPositionEnable AND btn_setPhaseUpperAxisPosition THEN
		FB_Set_PhaseUpperAxisPosition.ValueSet:=PhaseUpperSetValue;
		A_SetPhaseUpperAxisPosition();
END_IF
(************SetAxisPosition-GAP*********************)
IF  NOT USELinearEncoder AND setPhaseLowerAxisPositionEnable AND btn_setPhaseLowerAxisPosition THEN
		FB_Set_PhaseLowerAxisPosition.ValueSet:=PhaseLowerSetValue;
		A_SetPhaseLowerAxisPosition();
END_IF
(*******模式选择******)
IF SafePLCRunOK OR Simulation THEN
	IF pbSingleCarrierMode AND NOT pbTaperMode AND NOT pbGapMode AND NOT pbDebugMode AND NOT pbBCGapMode AND NOT pbUserMode THEN
		SingleCarrierMode();
	ELSIF pbTaperMode  AND NOT pbSingleCarrierMode AND NOT pbGapMode  AND NOT pbDebugMode AND NOT pbBCGapMode AND NOT pbUserMode THEN
		TaperMode();
	ELSIF pbGapMode AND  NOT pbSingleCarrierMode AND NOT pbTaperMode  AND NOT pbDebugMode AND NOT pbBCGapMode AND NOT pbUserMode THEN
		GapMode();
	ELSIF pbDebugMode AND NOT pbGapMode AND NOT pbSingleCarrierMode AND NOT pbTaperMode AND NOT pbBCGapMode  AND NOT pbUserMode THEN
		DebugMode();
	ELSIF pbBCGapMode AND NOT pbGapMode AND NOT pbSingleCarrierMode AND NOT pbTaperMode AND NOT pbDebugMode AND NOT pbUserMode THEN
		BCGapMode();
	ELSIF pbUserMode AND NOT pbGapMode AND NOT pbSingleCarrierMode AND NOT pbTaperMode AND NOT pbDebugMode AND NOT pbBCGapMode THEN
		UserMode();
	END_IF
END_IF
(*******Led Show******)
fb_led_Show();
(*******Check Power status******)
FB_Power(Check:=TRUE);
st_Power:=FB_Power.PowerState;
(******Check Couple Status*****)
FB_CheckCoupleStatus(Check:=TRUE);
st_Couple:=FB_CheckCoupleStatus.CoupleState;

(*********RS232*********************)
BackgroundEL();

(*获取温度传感器数据*)
//A_GetTemperatureSensorsData();

(*设置position bias*)
IF loadParametersDone AND (DriveStatus=1 OR simulation) THEN 
	A_SetLinearEncoderPositionBias();
END_IF
(*检查硬急停状态，包括安全限位、柜门急停、手持急停*)
A_CheckHardwareEmergencyStopStatus();
IF NOT simulation THEN
	A_GetDriverStatus();
END_IF
(*IDControlReady*)
IF ((DriveStatus<>0 AND SafePLCRunOK) OR simulation) AND NOT Error THEN
	IDControlReady:=TRUE;
ELSE
	IDControlReady:=FALSE;
END_IF

(*IOC Start*)
IF SafePLCRunOK OR simulation THEN
	bExe_load_Prog:=TRUE;
	A_LoadOpcIocShellExe();
END_IF

(*RestartDrivers*)
A_RestartDrivers();

(*检查光栅读数是否在范围内*)
A_CheckLinearEncoder();


(*A_LEHeartBeatMonitor*)
IF LEHeartBeatMonitorFunctionOn THEN
	A_LEHeartBeatMonitor();
END_IF
(************SetMotorAxisPosition*********************)
//IDControl 1s after
fb_ton5_2.IN:=IDControlReady;
fb_ton5_2.PT:=T#1S;
fb_ton5_2();
IF fb_ton5_2.Q THEN
	btn_SetMotorAxisPosition:=TRUE;
	btn_SetPhaseUpperMotorAxisPosition:=TRUE;
	btn_SetPhaseLowerMotorAxisPosition:=TRUE;
END_IF
IF  USELinearEncoder AND btn_SetMotorAxisPosition THEN
	IF NOT SetMotorAxisPositionDone THEN
		FB_Set_MotorAxisPosition.ValueSet_LeftTop:=Pos_LeftTopLin;
		FB_Set_MotorAxisPosition.ValueSet_RightTop:=Pos_RightTopLin;
		FB_Set_MotorAxisPosition.ValueSet_LeftBottom:=Pos_LeftBottomLin;
		FB_Set_MotorAxisPosition.ValueSet_RightBottom:=Pos_RightBottomLin;
		A_SetMotorAxisPosition();
	END_IF
END_IF
IF  USELinearEncoder AND btn_SetPhaseUpperMotorAxisPosition THEN
	IF NOT SetPhaseUpperMotorAxisPositionDone THEN
		FB_Set_PhaseUpperMotorAxisPosition.ValueSet:=Pos_PhaseUpperLin;
		A_SetPhaseUpperMotorAxisPosition();
	END_IF
END_IF
IF  USELinearEncoder AND btn_SetPhaseLowerMotorAxisPosition THEN
	IF NOT SetPhaseLowerMotorAxisPositionDone THEN
		FB_Set_PhaseLowerMotorAxisPosition.ValueSet:=Pos_PhaseLowerLin;
		A_SetPhaseLowerMotorAxisPosition();
	END_IF
END_IF
(*A_MonitorMotorAndLE*)
IF MonitorMotorAndLEFunctionOn AND SetMotorAxisPositionDone 
	AND SetPhaseUpperMotorAxisPositionDone AND SetPhaseLowerMotorAxisPositionDone THEN
	A_MonitorMotorAndLE();
END_IF
(*A_CheckMaxVelocity*)
A_CheckMaxVelocity();
(**)
A_GetMotorTemperature();

A_PolarStatus();

ACTION A_CheckHardwareEmergencyStopStatus:
IF 	NOT KS_LeftTop_Far_Contact1 OR
	NOT KS_LeftTop_Far_Contact2 OR
	NOT KS_RightTop_Far_Contact1 OR
	NOT KS_RightTop_Far_Contact2 OR
	NOT KS_LeftBottom_Far_Contact1 OR
	NOT KS_LeftBottom_Far_Contact2 OR
	NOT KS_RightBottom_Far_Contact1 OR
	NOT KS_RightBottom_Far_Contact2 OR
	NOT KS_PhaseUpper_Exit_Contact1 OR
	NOT KS_PhaseUpper_Exit_Contact2 OR
	NOT KS_PhaseLower_Exit_Contact1 OR
	NOT KS_PhaseLower_Exit_Contact2 OR
	
	NOT KS_LeftTop_Near_Contact1 OR
	NOT KS_LeftTop_Near_Contact2 OR
	NOT KS_RightTop_Near_Contact1 OR
	NOT KS_RightTop_Near_Contact2 OR
	NOT KS_LeftBottom_Near_Contact1 OR
	NOT KS_LeftBottom_Near_Contact2 OR
	NOT KS_RightBottom_Near_Contact1 OR
	NOT KS_RightBottom_Near_Contact2 OR
	NOT KS_PhaseUpper_Entrance_Contact1 OR
	NOT KS_PhaseUpper_Entrance_Contact2 OR
	NOT KS_PhaseLower_Entrance_Contact1 OR
	NOT KS_PhaseLower_Entrance_Contact2 OR
(*E-STOP*)
	NOT KS_CabinetEmergency_contact1 OR
	NOT KS_CabinetEmergency_contact2 OR
	NOT KS_handEmergency1_Contact1 OR
	NOT KS_handEmergency1_Contact2 OR
	NOT KS_handEmergency2_Contact1 OR
	NOT KS_handEmergency2_Contact2 OR
	NOT KS_softEmergency2_Contact THEN
	Hardware_EmergencyStop:=FALSE;
ELSE
	Hardware_EmergencyStop:=TRUE;
END_IF
END_ACTION

ACTION A_CheckKillSwitch:
IF simulation THEN
	//EL1904-1
	KS_LeftTop_Far_Contact1:=TRUE;
	KS_LeftTop_Far_Contact2:=TRUE;
	KS_LeftTop_Near_Contact1:=TRUE;
	KS_LeftTop_Near_Contact2:=TRUE;
	//EL1904-2
	KS_RightTop_Far_Contact1:=TRUE;
	KS_RightTop_Far_Contact2:=TRUE;
	KS_RightTop_Near_Contact1:=TRUE;
	KS_RightTop_Near_Contact2:=TRUE;
	//EL1904-3
	KS_LeftBottom_Far_Contact1:=TRUE;
	KS_LeftBottom_Far_Contact2:=TRUE;
	KS_LeftBottom_Near_Contact1:=TRUE;
	KS_LeftBottom_Near_Contact2:=TRUE;
	//EL1904-4
	KS_RightBottom_Far_Contact1:=TRUE;
	KS_RightBottom_Far_Contact2:=TRUE;
	KS_RightBottom_Near_Contact1:=TRUE;
	KS_RightBottom_Near_Contact2:=TRUE;
	//EL1904-5
	KS_PhaseUpper_Exit_Contact1:=TRUE;
	KS_PhaseUpper_Exit_Contact2:=TRUE;
	KS_PhaseUpper_Entrance_Contact1:=TRUE;
	KS_PhaseUpper_Entrance_Contact2:=TRUE;
	//EL1904-6
	KS_PhaseLower_Exit_Contact1:=TRUE;
	KS_PhaseLower_Exit_Contact2:=TRUE;
	KS_PhaseLower_Entrance_Contact1:=TRUE;
	KS_PhaseLower_Entrance_Contact2:=TRUE;
	//EL1904-7
	(*E-STOP*)
	(*柜门急停*)
	KS_CabinetEmergency_contact1:=TRUE;
	KS_CabinetEmergency_contact2:=TRUE;
	(*手持急停-1*)
	KS_handEmergency1_Contact1:=TRUE;
	KS_handEmergency1_Contact2:=TRUE;
	//EL1904-8
	(*手持急停-2*)
	KS_handEmergency2_Contact1:=TRUE;
	KS_handEmergency2_Contact2:=TRUE;
	
	KS_softEmergency2_Contact:=TRUE;
	AX5805_ErrorAsk:=TRUE;
ELSE
	//EL1904-1
	KS_LeftTop_Far_Contact1:=EL1904[1];//c1
	KS_LeftTop_Far_Contact2:=EL1904[2];//c2
	KS_LeftTop_Near_Contact1:=EL1904[3];//c3
	KS_LeftTop_Near_Contact2:=EL1904[4];//c4
	//EL1904-2
	KS_RightTop_Far_Contact1:=EL1904[5];
	KS_RightTop_Far_Contact2:=EL1904[6];
	KS_RightTop_Near_Contact1:=EL1904[7];
	KS_RightTop_Near_Contact2:=EL1904[8];
	//EL1904-3
	KS_LeftBottom_Far_Contact1:=EL1904[9];
	KS_LeftBottom_Far_Contact2:=EL1904[10];
	KS_LeftBottom_Near_Contact1:=EL1904[11];
	KS_LeftBottom_Near_Contact2:=EL1904[12];
	//EL1904-4
	KS_RightBottom_Far_Contact1:=EL1904[13];
	KS_RightBottom_Far_Contact2:=EL1904[14];
	KS_RightBottom_Near_Contact1:=EL1904[15];
	KS_RightBottom_Near_Contact2:=EL1904[16];	
	//EL1904-5
	KS_PhaseUpper_Exit_Contact1:=EL1904[17];
	KS_PhaseUpper_Exit_Contact2:=EL1904[18];
	KS_PhaseUpper_Entrance_Contact1:=EL1904[19];
	KS_PhaseUpper_Entrance_Contact2:=EL1904[20];
	//EL1904-6
	KS_PhaseLower_Exit_Contact1:=EL1904[21];
	KS_PhaseLower_Exit_Contact2:=EL1904[22];
	KS_PhaseLower_Entrance_Contact1:=EL1904[23];
	KS_PhaseLower_Entrance_Contact2:=EL1904[24];
	//EL1904-7
	(*E-STOP*)
	(*柜门急停*)
	KS_CabinetEmergency_contact1:=EL1904[25];
	KS_CabinetEmergency_contact2:=EL1904[26];
	(*手持急停-1*)
	KS_handEmergency1_Contact1:=EL1904[27];
	KS_handEmergency1_Contact2:=EL1904[28];
	//EL1904-8
	(*手持急停-2*)
	KS_handEmergency2_Contact1:=EL1904[29];
	KS_handEmergency2_Contact2:=EL1904[30];
	
	KS_softEmergency2_Contact:=EL1904[31];
	AX5805_ErrorAsk:=EL1904[32];

END_IF
END_ACTION

ACTION A_CheckLimitSwitch:
(*******1.´ÓIO»ñÈ¡ÏÞÎ»×´Ì¬******)
(*
IF simulation THEN
	(**)
	LS_LeftTop_Far:=TRUE;
	LS_LeftTop_Near:=TRUE;
	LS_RightTop_Far:=TRUE;
	LS_RightTop_Near:=TRUE;
	LS_LeftBottom_Far:=TRUE;
	LS_LeftBottom_Near:=TRUE;
	LS_RightBottom_Far:=TRUE;
	LS_RightBottom_Near:=TRUE;
	LS_PhaseUpper_Entrance:=TRUE;
	LS_PhaseUpper_Exit:=TRUE;
	LS_PhaseLower_Entrance:=TRUE;
	LS_PhaseLower_Exit:=TRUE;
	
ELSE
	LS_LeftTop_Far :=el1808_D1[1];
	LS_LeftTop_Near:=el1808_D1[3];
	LS_RightTop_Far:=el1808_D1[2];
	LS_RightTop_Near:=el1808_D1[4];
	LS_LeftBottom_Far:=el1808_D1[7];
	LS_LeftBottom_Near:=el1808_D1[5];
	LS_RightBottom_Far:=el1808_D1[8];
	LS_RightBottom_Near:=el1808_D1[6];
	LS_PhaseUpper_Entrance:=el1808_D2[1];
	LS_PhaseUpper_Exit:=el1808_D2[2];
	LS_PhaseLower_Entrance:=el1808_D2[3];
	LS_PhaseLower_Exit:=el1808_D2[4];
END_IF

*)
(*
	LS_LeftTop_Top:=TRUE;
	LS_LeftTop_Bottom:=TRUE;
	LS_RightTop_Top:=TRUE;
	LS_RightTop_Bottom:=TRUE;
	LS_LeftBottom_Top:=TRUE;
	LS_LeftBottom_Bottom:=TRUE;
	LS_RightBottom_Top:=TRUE;
	LS_RightBottom_Bottom:=TRUE;
*)
(******2.TopÏÞÎ»»òÕßBottomÏÞÎ»ÓÐÒ»¸ö´¥·¢£¬È«¾Ö±äÁ¿¡£¸øMC_POWERÓÃÓÚ·½Ïò¿ØÖÆ£¬ÓÐÒ»¸öÏÞÎ»Îª´¥·¢ÎªFALSE£¬ÔòUnreach_LSÎªFALSE******)
Unreach_LS_Far:=LS_LeftTop_Far AND LS_RightTop_Far AND LS_LeftBottom_Far AND LS_RightBottom_Far;
Unreach_LS_Near:=LS_LeftTop_Near AND LS_RightTop_Near AND LS_LeftBottom_Near AND LS_RightBottom_Near;
(**************************ÏòTopÔË¶¯Ê±£¬´¥ÅöBottomÏÞÎ»¿ª¹Ø£¬»òÕßÏà·´£¬ESTOP**************************************)
(*
IF LeftTopLin.Status.Moving AND Velo_LeftTopLin>0 THEN
	IF NOT Unreach_LS_Bottom THEN
		Error:=TRUE;
		ErrorID:=61;
		FB_PlcEmergencyStop();
	END_IF
ELSIF LeftTopLin.Status.Moving AND Velo_LeftTopLin<0 THEN
	IF NOT Unreach_LS_Top THEN
		Error:=TRUE;
		ErrorID:=62;
		FB_PlcEmergencyStop();
	END_IF
ELSIF RightTopLin.Status.Moving AND Velo_RightTopLin>0 THEN
	IF NOT Unreach_LS_Bottom THEN
		Error:=TRUE;
		ErrorID:=63;
		FB_PlcEmergencyStop();
	END_IF
ELSIF RightTopLin.Status.Moving AND Velo_RightTopLin<0 THEN
	IF NOT  Unreach_LS_Top THEN
		Error:=TRUE;
		ErrorID:=64;
		FB_PlcEmergencyStop();
	END_IF
ELSIF LeftBottomLin.Status.Moving AND Velo_LeftBottomLin>0 THEN
	IF NOT Unreach_LS_Bottom THEN
		Error:=TRUE;
		ErrorID:=65;
		FB_PlcEmergencyStop();
	END_IF
ELSIF LeftBottomLin.Status.Moving AND Velo_LeftBottomLin<0 THEN
	IF NOT Unreach_LS_Top THEN
		Error:=TRUE;
		ErrorID:=66;
		FB_PlcEmergencyStop();
	END_IF
ELSIF RightBottomLin.Status.Moving AND Velo_RightBottomLin>0 THEN
	IF NOT Unreach_LS_Bottom THEN
		Error:=TRUE;
		ErrorID:=67;
		FB_PlcEmergencyStop();
	END_IF
ELSIF RightBottomLin.Status.Moving AND Velo_RightBottomLin<0 THEN
	IF NOT Unreach_LS_Top THEN
		Error:=TRUE;
		ErrorID:=68;
		FB_PlcEmergencyStop();
	END_IF
END_IF
*)
(*
(******3.ÓÐÒ»¸öÏÞÎ»´¥·¢£¬ delayÊ±¼äºó£¬¼à²âÖáÊÇ·ñÔÚÍ£Ö¹×´Ì¬£¬ÈôÃ»ÓÐ£¬Emergency AND PowerOff******)
IF NOT Unreach_LS_Top OR NOT Unreach_LS_Bottom THEN
	fb_ton.IN:=TRUE;
END_IF
IF fb_ton.Q THEN
	IF LeftTopLin.Status.Moving OR RightTopLin.Status.Moving OR LeftBottomLin.Status.Moving OR RightBottomLin.Status.Moving THEN
		FB_PlcEmergencyStop();
		fb_ton.IN:=FALSE;
		Error:=TRUE;
		EStopTrig:=TRUE;
		ErrorID:=1;
		(*FB_Power_Off(Execute:=TRUE);*)
	END_IF
END_IF

(*******4.µ¥ÖáÉÏÏÂÏÞÎ»¾ùÎªFALSEÊ±£¬ÏÞÎ»´íÎó£¬Emergency*******)
IF (NOT LS_LeftTop_Top AND NOT LS_LeftTop_Bottom) OR  (NOT  LS_RightTop_Top AND NOT LS_RightTop_Bottom)
		OR (NOT LS_LeftBottom_Top AND NOT LS_LeftBottom_Bottom) OR (NOT LS_RightBottom_Top AND NOT LS_RightBottom_Bottom) THEN
	(*FB_Plc_EmergencyStop();*)
	Error:=TRUE;
	EStopTrig:=TRUE;
	ErrorID:=2;
END_IF
*)
END_ACTION

ACTION A_CheckLinearEncoder:
//LE Protection Position
min_UserLEProtectionGapPosition:=min_UserGapPositionNew-min_ThresholdGapSoft2LEProtection;//回程误差有0.1mm
max_UserLEProtectionGapPosition:=max_UserGapPositionNew+max_ThresholdGapSoft2LEProtection;
//如果没有使用光栅、或者光栅参数没设置好，则不检查光栅位置
IF NOT USELinearEncoder OR NOT PositionBiasDone THEN
	RETURN;
END_IF
IF Pos_LeftTopLin <=0 THEN
	ErrorID:=1101;
	Error:=TRUE;
	ErrorDescription:='Pos_LeftTopLin <=0';
	FB_PlcEmergencyStop();
	LED_Error:=TRUE;
END_IF
IF Pos_RightTopLin <=0 THEN
	ErrorID:=1102;
	Error:=TRUE;
	ErrorDescription:='Pos_RightTopLin <=0';
	FB_PlcEmergencyStop();
	LED_Error:=TRUE;
END_IF
IF Pos_LeftBottomLin <=0 THEN
	ErrorID:=1103;
	Error:=TRUE;
	ErrorDescription:='Pos_LeftBottomLin <=0';
	FB_PlcEmergencyStop();
	LED_Error:=TRUE;
END_IF
IF Pos_RightBottomLin <=0 THEN
	ErrorID:=1104;
	Error:=TRUE;
	ErrorDescription:='Pos_RightBottomLin <=0';
	FB_PlcEmergencyStop();
	LED_Error:=TRUE;
END_IF

//
IF Pos_LeftTopLin >max_UserLEProtectionGapPosition/2 THEN
	ErrorID:=1105;
	Error:=TRUE;
	ErrorDescription:='Pos_LeftTopLin >max_UserLEProtectionGapPosition/2';
	FB_PlcEmergencyStop();
	LED_Error:=TRUE;
END_IF
IF Pos_RightTopLin >max_UserLEProtectionGapPosition/2 THEN
	ErrorID:=1106;
	Error:=TRUE;
	ErrorDescription:='Pos_RightTopLin>max_UserLEProtectionGapPosition/2';
	FB_PlcEmergencyStop();
	LED_Error:=TRUE;
END_IF
IF Pos_LeftBottomLin >max_UserLEProtectionGapPosition/2 THEN
	ErrorID:=1107;
	Error:=TRUE;
	ErrorDescription:='Pos_LeftBottomLin >max_UserLEProtectionGapPosition/2';
	FB_PlcEmergencyStop();
	LED_Error:=TRUE;
END_IF
IF Pos_RightBottomLin >max_UserLEProtectionGapPosition/2 THEN
	ErrorID:=1108;
	Error:=TRUE;
	ErrorDescription:='Pos_RightBottomLin >max_UserLEProtectionGapPosition/2';
	FB_PlcEmergencyStop();
	LED_Error:=TRUE;
END_IF


IF Pos_LeftTopLin <min_UserLEProtectionGapPosition/2 THEN
	ErrorID:=1109;
	Error:=TRUE;
	ErrorDescription:='Pos_LeftTopLin <min_UserLEProtectionGapPosition/2';
	FB_PlcEmergencyStop();
	LED_Error:=TRUE;
END_IF
IF Pos_RightTopLin <min_UserLEProtectionGapPosition/2 THEN
	ErrorID:=1110;
	Error:=TRUE;
	ErrorDescription:='Pos_RightTopLin<min_UserLEProtectionGapPosition/2';
	FB_PlcEmergencyStop();
	LED_Error:=TRUE;
END_IF
IF Pos_LeftBottomLin <min_UserLEProtectionGapPosition/2 THEN
	ErrorID:=1111;
	Error:=TRUE;
	ErrorDescription:='Pos_LeftBottomLin <min_UserLEProtectionGapPosition';
	FB_PlcEmergencyStop();
	LED_Error:=TRUE;
END_IF
IF Pos_RightBottomLin <min_UserLEProtectionGapPosition/2 THEN
	ErrorID:=1112;
	Error:=TRUE;
	ErrorDescription:='Pos_RightBottomLin <min_UserLEProtectionGapPosition';
	FB_PlcEmergencyStop();
	LED_Error:=TRUE;
END_IF
//
//PhaseUpper方向
//
min_UserLEProtectionPhaseUpperPosition:=min_UserPhaseUpperPositionNew-min_ThresholdPhaseUpperSoft2LEProtection;//回程误差有0.1mm
max_UserLEProtectionPhaseUpperPosition:=max_UserPhaseUpperPositionNew+max_ThresholdPhaseUpperSoft2LEProtection;
IF Pos_PhaseUpperLin >max_UserLEProtectionPhaseUpperPosition THEN
	ErrorID:=1113;
	Error:=TRUE;
	ErrorDescription:=' Pos_PhaseUpperLin >max_UserLEProtectionPhaseUpperPosition';
	FB_PlcEmergencyStop();
	LED_Error:=TRUE;
END_IF
IF Pos_PhaseUpperLin < min_UserLEProtectionPhaseUpperPosition THEN
	ErrorID:=1114;
	Error:=TRUE;
	ErrorDescription:=' Pos_PhaseUpperLin >< min_UserLEProtectionPhaseUpperPosition';
	FB_PlcEmergencyStop();
	LED_Error:=TRUE;
END_IF
//
//PhaseLower方向
//
min_UserLEProtectionPhaseLowerPosition:=min_UserPhaseLowerPositionNew-min_ThresholdPhaseLowerSoft2LEProtection;//回程误差有0.1mm
max_UserLEProtectionPhaseLowerPosition:=max_UserPhaseLowerPositionNew+max_ThresholdPhaseLowerSoft2LEProtection;
IF Pos_PhaseLowerLin >max_UserLEProtectionPhaseLowerPosition THEN
	ErrorID:=1115;
	Error:=TRUE;
	ErrorDescription:=' Pos_PhaseLowerLin >max_UserLEProtectionPhaseLowerPosition';
	FB_PlcEmergencyStop();
	LED_Error:=TRUE;
END_IF
IF Pos_PhaseLowerLin < min_UserLEProtectionPhaseLowerPosition THEN
	ErrorID:=1116;
	Error:=TRUE;
	ErrorDescription:=' Pos_PhaseLowerLin < min_UserLEProtectionPhaseLowerPosition';
	FB_PlcEmergencyStop();
	LED_Error:=TRUE;
END_IF
END_ACTION

ACTION A_CheckMaxVelocity:
IF NOT USELinearEncoder OR NOT PositionBiasDone OR NOT IDControlReady THEN
	RETURN;
END_IF
IF NOT st_Power THEN
	RETURN;
END_IF
//Monitoring Motor and LE Position/Velocity
MaxVelocityGlobalVelocity:=MAX(max_UserGapVelocityNew,max_UserTaperVelocityNew,UserMode.max_SS_StepVelocity,
			UserMode.Global_ChainProtection_MPS_MoveVelocity,UserMode.Global_ChainProtection_EPS_MoveVelocity);
IF 	ABS(Velo_LeftTopLin) > MaxVelocityGlobalVelocity*1.1/2 THEN
	ErrorID:=7001;
	Error:=TRUE;
	ErrorDescription:='ABS(Velo_LeftTopLin) > MaxVelocityGlobalVelocity*1.1/2';
	FB_PlcEmergencyStop();
	LED_Error:=TRUE;
END_IF
IF 	ABS(Velo_LeftTopMotor) > MaxVelocityGlobalVelocity*1.1/2 THEN
	ErrorID:=7002;
	Error:=TRUE;
	ErrorDescription:='ABS(Velo_LeftTopMotor) > MaxVelocityGlobalVelocity*1.1/2';
	FB_PlcEmergencyStop();
	LED_Error:=TRUE;
END_IF
IF 	ABS(Velo_RightTopLin) > MaxVelocityGlobalVelocity*1.1/2 THEN
	ErrorID:=7003;
	Error:=TRUE;
	ErrorDescription:='ABS(Velo_RightTopLin) > MaxVelocityGlobalVelocity*1.1/2';
	FB_PlcEmergencyStop();
	LED_Error:=TRUE;
END_IF
IF 	ABS(Velo_RightTopMotor) > MaxVelocityGlobalVelocity*1.1/2 THEN
	ErrorID:=7004;
	Error:=TRUE;
	ErrorDescription:='ABS(Velo_RightTopMotor) > MaxVelocityGlobalVelocity*1.1/2';
	FB_PlcEmergencyStop();
	LED_Error:=TRUE;
END_IF
IF 	ABS(Velo_LeftBottomLin) > MaxVelocityGlobalVelocity*1.1/2 THEN
	ErrorID:=7005;
	Error:=TRUE;
	ErrorDescription:='ABS(Velo_LeftBottomLin) > MaxVelocityGlobalVelocity*1.1/2';
	FB_PlcEmergencyStop();
	LED_Error:=TRUE;
END_IF
IF 	ABS(Velo_LeftBottomMotor) > MaxVelocityGlobalVelocity*1.1/2 THEN
	ErrorID:=7006;
	Error:=TRUE;
	ErrorDescription:='ABS(Velo_LeftBottomMotor) > MaxVelocityGlobalVelocity*1.1/2';
	FB_PlcEmergencyStop();
	LED_Error:=TRUE;
END_IF
IF 	ABS(Velo_RightBottomLin) > MaxVelocityGlobalVelocity*1.1/2 THEN
	ErrorID:=7007;
	Error:=TRUE;
	ErrorDescription:='ABS(Velo_RightBottomLin) > MaxVelocityGlobalVelocity*1.1/2';
	FB_PlcEmergencyStop();
	LED_Error:=TRUE;
END_IF
IF 	ABS(Velo_RightBottomMotor) > MaxVelocityGlobalVelocity*1.1/2 THEN
	ErrorID:=7008;
	Error:=TRUE;
	ErrorDescription:='ABS(Velo_RighBottomMotor) > MaxVelocityGlobalVelocity*1.1/2';
	FB_PlcEmergencyStop();
	LED_Error:=TRUE;
END_IF
(*
IF 	ABS(Velo_PhaseUpperLin) > MaxVelocityGlobalVelocity*1.1/2 THEN
	ErrorID:=7005;
	Error:=TRUE;
	ErrorDescription:='ABS(Velo_PhaseUpperLin) > MaxVelocityGlobalVelocity*1.1/2';
	FB_PlcEmergencyStop();
	LED_Error:=TRUE;
END_IF
IF 	ABS(Velo_PhaseUpperMotor) > MaxVelocityGlobalVelocity*1.1/2 THEN
	ErrorID:=7006;
	Error:=TRUE;
	ErrorDescription:='ABS(Velo_PhaseUpperMotor) > MaxVelocityGlobalVelocity*1.1/2';
	FB_PlcEmergencyStop();
	LED_Error:=TRUE;
END_IF
IF 	ABS(Velo_PhaseLowerLin) > MaxVelocityGlobalVelocity*1.1/2 THEN
	ErrorID:=7007;
	Error:=TRUE;
	ErrorDescription:='ABS(Velo_PhaseLowerLin) > MaxVelocityGlobalVelocity*1.1/2';
	FB_PlcEmergencyStop();
	LED_Error:=TRUE;
END_IF
IF 	ABS(Velo_PhaseLowerMotor) > MaxVelocityGlobalVelocity*1.1/2 THEN
	ErrorID:=7008;
	Error:=TRUE;
	ErrorDescription:='ABS(Velo_RighBottomMotor) > MaxVelocityGlobalVelocity*1.1/2';
	FB_PlcEmergencyStop();
	LED_Error:=TRUE;
END_IF
*)
END_ACTION

ACTION A_GetDriverStatus:
//
//DriveMessage/Drive Number/Gear number/feedback2 direction
//
IF bReloadDriveDiagMessageAndNumber THEN
	m_GetDriveStatusState:=0;
	bReloadDriveDiagMessageAndNumber:=FALSE;
END_IF
GetDriveStatusTON(PT:=T#1S);
GetDriveStatusTON2(PT:=T#0.1S);
A_GetDriverStatusMC();
CASE m_GetDriveStatusState OF
	0:
		GetDriveStatusTON.IN:=TRUE;
		m_GetDriveStatusState:=1;
	1:
		IF GetDriveStatusTON.Q THEN
			bDriveDiagMessageAndNumber:=TRUE;
			m_GetDriveStatusState:=2;
		END_IF
	2:
		GetDriveStatusTON.IN:=FALSE;
		DriveDiagMessage_LeftTop:=fb_SoEReadDiagMessage_LeftTop.sDiagMessage.strData;
		DriveDiagMessage_RightTop:=fb_SoEReadDiagMessage_RightTop.sDiagMessage.strData;
		DriveDiagMessage_LeftBottom:=fb_SoEReadDiagMessage_LeftBottom.sDiagMessage.strData;
		DriveDiagMessage_RightBottom:=fb_SoEReadDiagMessage_RightBottom.sDiagMessage.strData;
		DriveDiagMessage_PhaseUpper:=fb_SoEReadDiagMessage_PhaseUpper.sDiagMessage.strData;
		DriveDiagMessage_PhaseLower:=fb_SoEReadDiagMessage_PhaseLower.sDiagMessage.strData;
		//
		DriveDiagNumber_LeftTop:=FB_SoEReadDiagNumber_LeftTop.iDiagNumber;
		DriveDiagNumber_RightTop:=FB_SoEReadDiagNumber_RightTop.iDiagNumber;
		DriveDiagNumber_LeftBottom:=FB_SoEReadDiagNumber_LeftBottom.iDiagNumber;
		DriveDiagNumber_RightBottom:=FB_SoEReadDiagNumber_RightBottom.iDiagNumber;
		DriveDiagNumber_PhaseUpper:=FB_SoEReadDiagNumber_PhaseUpper.iDiagNumber;
		DriveDiagNumber_PhaseLower:=FB_SoEReadDiagNumber_PhaseLower.iDiagNumber;
		//
		GearNumeratorGet_LeftTop:=st_p182_LeftTop.Feedback_2_geat_numerator;
		GearNumeratorGet_RightTop:=st_p182_RightTop.Feedback_2_geat_numerator;
		GearNumeratorGet_LeftBottom:=st_p182_LeftBottom.Feedback_2_geat_numerator;
		GearNumeratorGet_RightBottom:=st_p182_RightBottom.Feedback_2_geat_numerator;
		GearNumeratorGet_PhaseUpper:=st_p182_PhaseUpper.Feedback_2_geat_numerator;
		GearNumeratorGet_PhaseLower:=st_p182_PhaseLower.Feedback_2_geat_numerator;
		//
		GearDenominatorGet_LeftTop:=st_p183_LeftTop.Feedback_2_geat_denominator;
		GearDenominatorGet_RightTop:=st_p183_RightTop.Feedback_2_geat_denominator;
		GearDenominatorGet_LeftBottom:=st_p183_LeftBottom.Feedback_2_geat_denominator;
		GearDenominatorGet_RightBottom:=st_p183_RightBottom.Feedback_2_geat_denominator;
		GearDenominatorGet_PhaseUpper:=st_p183_PhaseUpper.Feedback_2_geat_denominator;
		GearDenominatorGet_PhaseLower:=st_p183_PhaseLower.Feedback_2_geat_denominator;
		//
		Feedback2directionGet_LeftTop:=st_p180_LeftTop.Feedback_direction;
		Feedback2directionGet_RightTop:=st_p180_RightTop.Feedback_direction;
		Feedback2directionGet_LeftBottom:=st_p180_LeftBottom.Feedback_direction;
		Feedback2directionGet_RightBottom:=st_p180_RightBottom.Feedback_direction;
		Feedback2directionGet_PhaseUpper:=st_p180_PhaseUpper.Feedback_direction;
		Feedback2directionGet_PhaseLower:=st_p180_PhaseLower.Feedback_direction;
		//
		IF 	NOT fb_SoEReadDiagMessage_LeftTop.bBusy
			AND NOT fb_SoEReadDiagMessage_RightTop.bBusy
			AND NOT fb_SoEReadDiagMessage_LeftBottom.bBusy
			AND NOT fb_SoEReadDiagMessage_RightBottom.bBusy 
			AND NOT fb_SoEReadDiagMessage_PhaseUpper.bBusy
			AND NOT fb_SoEReadDiagMessage_PhaseLower.bBusy 
			AND NOT FB_SoEReadDiagNumber_LeftTop.bBusy
			AND NOT FB_SoEReadDiagNumber_RightTop.bBusy
			AND NOT FB_SoEReadDiagNumber_LeftBottom.bBusy
			AND NOT FB_SoEReadDiagNumber_RightBottom.bBusy 
			AND NOT FB_SoEReadDiagNumber_PhaseUpper.bBusy
			AND NOT FB_SoEReadDiagNumber_PhaseLower.bBusy 
			AND NOT FB_SoERead_GearNumerator_LeftTop.bBusy 
			AND NOT FB_SoERead_GearNumerator_RightTop.bBusy 
			AND NOT FB_SoERead_GearNumerator_LeftBottom.bBusy 
			AND NOT FB_SoERead_GearNumerator_RightBottom.bBusy 
			AND NOT FB_SoERead_GearNumerator_PhaseUpper.bBusy 
			AND NOT FB_SoERead_GearNumerator_PhaseLower.bBusy 
			AND NOT FB_SoERead_GearDenominator_LeftTop.bBusy 
			AND NOT FB_SoERead_GearDenominator_RightTop.bBusy 
			AND NOT FB_SoERead_GearDenominator_LeftBottom.bBusy 
			AND NOT FB_SoERead_GearDenominator_RightBottom.bBusy 
			AND NOT FB_SoERead_GearDenominator_PhaseUpper.bBusy 
			AND NOT FB_SoERead_GearDenominator_PhaseLower.bBusy 
			AND NOT FB_SoERead_Feedback2direction_LeftTop.bBusy 
			AND NOT FB_SoERead_Feedback2direction_RightTop.bBusy  
			AND NOT FB_SoERead_Feedback2direction_LeftBottom.bBusy 
			AND NOT FB_SoERead_Feedback2direction_RightBottom.bBusy
			AND NOT FB_SoERead_Feedback2direction_PhaseUpper.bBusy 
			AND NOT FB_SoERead_Feedback2direction_PhaseLower.bBusy	THEN
				GetDriveStatusTON2.IN:=TRUE;
				IF GetDriveStatusTON2.Q THEN
					m_GetDriveStatusState:=88;
				END_IF
		END_IF
		IF 	fb_SoEReadDiagMessage_LeftTop.bError
			OR fb_SoEReadDiagMessage_RightTop.bError
			OR fb_SoEReadDiagMessage_LeftBottom.bError
			OR fb_SoEReadDiagMessage_RightBottom.bError
			OR fb_SoEReadDiagMessage_PhaseUpper.bError
			OR fb_SoEReadDiagMessage_PhaseLower.bError
			OR FB_SoEReadDiagNumber_LeftTop.bError
			OR FB_SoEReadDiagNumber_RightTop.bError
			OR FB_SoEReadDiagNumber_LeftBottom.bError
			OR FB_SoEReadDiagNumber_RightBottom.bError 
			OR FB_SoEReadDiagNumber_PhaseUpper.bError
			OR FB_SoEReadDiagNumber_PhaseLower.bError 
			OR FB_SoERead_GearNumerator_LeftTop.bError 
			OR FB_SoERead_GearNumerator_RightTop.bError 
			OR FB_SoERead_GearNumerator_LeftBottom.bError 
			OR FB_SoERead_GearNumerator_RightBottom.bError 
			OR FB_SoERead_GearNumerator_PhaseUpper.bError 
			OR FB_SoERead_GearNumerator_PhaseLower.bError 
			OR FB_SoERead_GearDenominator_LeftTop.bError 
			OR FB_SoERead_GearDenominator_RightTop.bError 
			OR FB_SoERead_GearDenominator_LeftBottom.bError 
			OR FB_SoERead_GearDenominator_RightBottom.bError 
			OR FB_SoERead_GearDenominator_PhaseUpper.bError 
			OR FB_SoERead_GearDenominator_PhaseLower.bError 
			OR FB_SoERead_Feedback2direction_LeftTop.bError 
			OR FB_SoERead_Feedback2direction_RightTop.bError 
			OR FB_SoERead_Feedback2direction_LeftBottom.bError 
			OR FB_SoERead_Feedback2direction_RightBottom.bError 
			OR FB_SoERead_Feedback2direction_PhaseUpper.bError 
			OR FB_SoERead_Feedback2direction_PhaseLower.bError 
		THEN
			m_GetDriveStatusState:=-100;
		END_IF
		
	88:
		bDriveDiagMessageAndNumber:=FALSE;
		A_GetDriverStatusMC();
		GetDriveStatusStateDone:=TRUE;
		GetDriveStatusStateError:=FALSE;
		//
		(*Drive Status*)
		//D012, Axis state machine: Control and power section ready,53266
		IF DriveDiagNumber_LeftTop=16#D012 AND DriveDiagNumber_RightTop=16#D012			
			AND DriveDiagNumber_LeftBottom=16#D012 AND DriveDiagNumber_RightBottom=16#D012
			AND DriveDiagNumber_PhaseUpper=16#D012 AND DriveDiagNumber_PhaseLower=16#D012 THEN
			DriveStatus:=1;
		//D013, Axis state machine: Axis in operation,53267
		ELSIF DriveDiagNumber_LeftTop=16#D013 AND DriveDiagNumber_RightTop=16#D013
			AND DriveDiagNumber_LeftBottom=16#D013 AND DriveDiagNumber_RightBottom=16#D013
			AND DriveDiagNumber_PhaseUpper=16#D013 AND DriveDiagNumber_PhaseLower=16#D013 THEN
			DriveStatus:=2;
		//D014，Axis state machine: Axis halt.53266和53267中间会经历这么一个状态，算正常状态
		ELSIF DriveDiagNumber_LeftTop=16#D014 AND DriveDiagNumber_RightTop=16#D014
			AND DriveDiagNumber_LeftBottom=16#D014 AND DriveDiagNumber_RightBottom=16#D014
			AND DriveDiagNumber_PhaseUpper=16#D014 AND DriveDiagNumber_PhaseLower=16#D014 THEN
			DriveStatus:=3;
		ELSE
			DriveStatus:=0;
		END_IF
		//
		//
		//	//check statusGet and status configured
		IF 	GearNumeratorGet_LeftTop<>GearNumeratorConfigured_LeftTop 
			OR GearNumeratorGet_RightTop<>GearNumeratorConfigured_RightTop
			OR GearNumeratorGet_LeftBottom<>GearNumeratorConfigured_LeftBottom 
			OR GearNumeratorGet_RightBottom<>GearNumeratorConfigured_RightBottom
			OR GearNumeratorGet_PhaseUpper<>GearNumeratorConfigured_PhaseUpper 
			OR GearNumeratorGet_PhaseLower<>GearNumeratorConfigured_PhaseLower
			OR GearDenominatorGet_LeftTop<>GearDenominatorConfigured_LeftTop 
			OR GearDenominatorGet_RightTop<>GearDenominatorConfigured_RightTop
			OR GearDenominatorGet_LeftBottom<>GearDenominatorConfigured_LeftBottom 
			OR GearDenominatorGet_RightBottom<>GearDenominatorConfigured_RightBottom
			OR GearDenominatorGet_PhaseUpper<>GearDenominatorConfigured_PhaseUpper 
			OR GearDenominatorGet_PhaseLower<>GearDenominatorConfigured_PhaseLower THEN
				bDriveDiagMessageAndNumber:=FALSE;
				A_GetDriverStatusMC();
				GetDriveStatusStateDone:=FALSE;
				GetDriveStatusStateError:=TRUE;
				Error:=TRUE;
				ErrorId:=1302;
				ErrorDescription:='gearParameters Error';
				Plc_EmergencyStop:=FALSE;
		END_IF
		IF USELinearEncoder THEN
			IF 	Feedback2directionGet_LeftTop<>Feedback2directionConfigured_LeftTop 
				OR Feedback2directionGet_RightTop<>Feedback2directionConfigured_RightTop
				OR Feedback2directionGet_LeftBottom<>Feedback2directionConfigured_LeftBottom 
				OR Feedback2directionGet_RightBottom<Feedback2directionConfigured_RightBottom 
				OR Feedback2directionGet_PhaseUpper<>Feedback2directionConfigured_PhaseUpper 
				OR Feedback2directionGet_PhaseLower<Feedback2directionConfigured_PhaseLower THEN
					bDriveDiagMessageAndNumber:=FALSE;
					A_GetDriverStatusMC();
					GetDriveStatusStateDone:=FALSE;
					GetDriveStatusStateError:=TRUE;
					Error:=TRUE;
					ErrorId:=1303;
					ErrorDescription:='fb2direction Error';
					Plc_EmergencyStop:=FALSE;
			END_IF 
		END_IF
		m_GetDriveStatusState:=0;
	-100:
		bDriveDiagMessageAndNumber:=FALSE;
		A_GetDriverStatusMC();
		GetDriveStatusStateDone:=FALSE;
		GetDriveStatusStateError:=TRUE;
		Error:=TRUE;
		ErrorId:=1301;
		ErrorDescription:='GetDriveStatusStateError';
END_CASE
END_ACTION

ACTION A_GetDriverStatusMC:
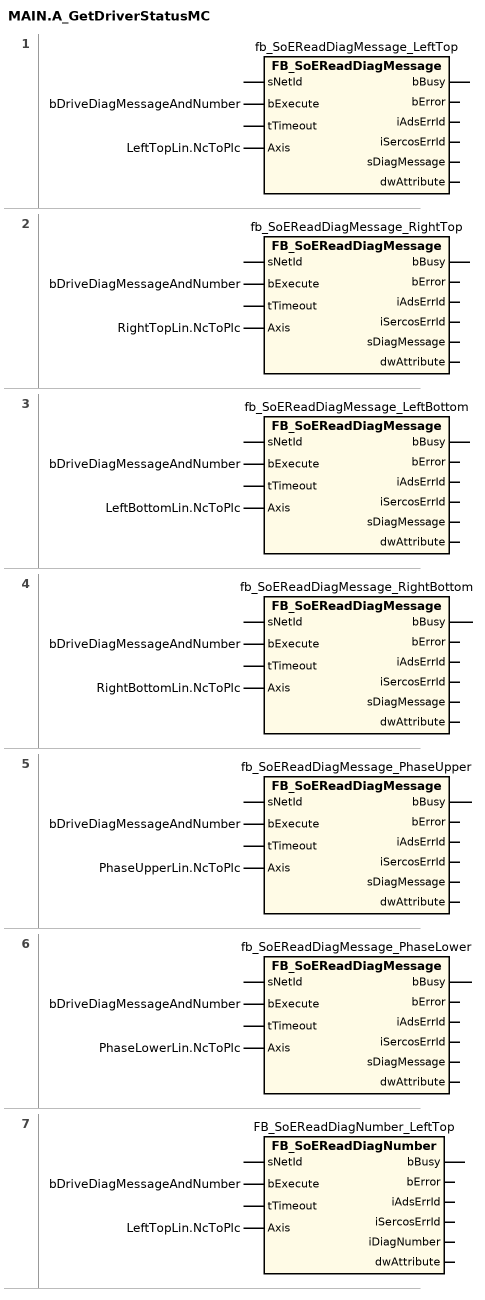
// NETWORK 1
fb_SoEReadDiagMessage_LeftTop(bExecute := bDriveDiagMessageAndNumber, Axis := LeftTopLin.NcToPlc); // FB_SoEReadDiagMessage

// NETWORK 2
fb_SoEReadDiagMessage_RightTop(bExecute := bDriveDiagMessageAndNumber, Axis := RightTopLin.NcToPlc); // FB_SoEReadDiagMessage

// NETWORK 3
fb_SoEReadDiagMessage_LeftBottom(bExecute := bDriveDiagMessageAndNumber, Axis := LeftBottomLin.NcToPlc); // FB_SoEReadDiagMessage

// NETWORK 4
fb_SoEReadDiagMessage_RightBottom(bExecute := bDriveDiagMessageAndNumber, Axis := RightBottomLin.NcToPlc); // FB_SoEReadDiagMessage

// NETWORK 5
fb_SoEReadDiagMessage_PhaseUpper(bExecute := bDriveDiagMessageAndNumber, Axis := PhaseUpperLin.NcToPlc); // FB_SoEReadDiagMessage

// NETWORK 6
fb_SoEReadDiagMessage_PhaseLower(bExecute := bDriveDiagMessageAndNumber, Axis := PhaseLowerLin.NcToPlc); // FB_SoEReadDiagMessage

// NETWORK 7
FB_SoEReadDiagNumber_LeftTop(bExecute := bDriveDiagMessageAndNumber, Axis := LeftTopLin.NcToPlc); // FB_SoEReadDiagNumber

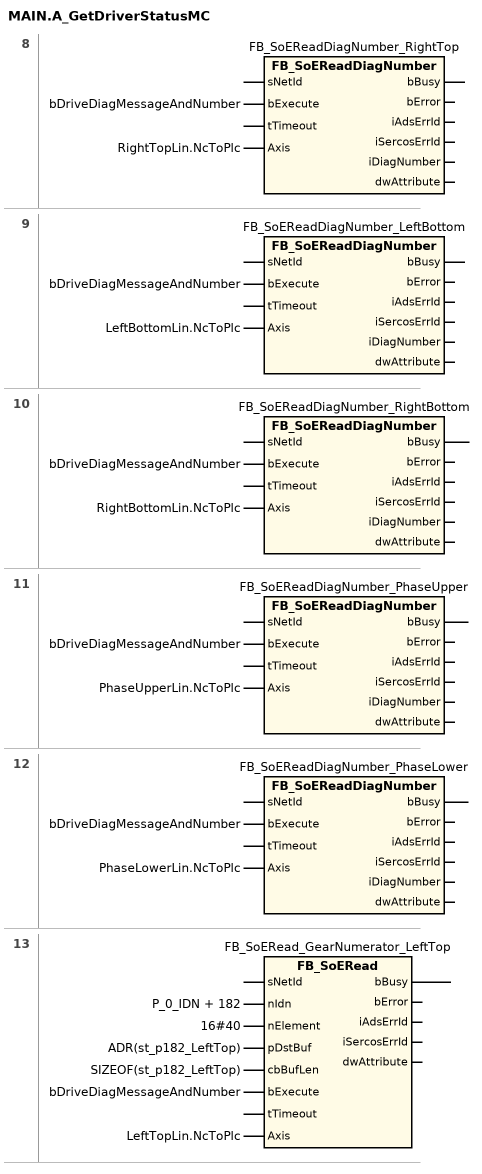
// NETWORK 8
FB_SoEReadDiagNumber_RightTop(bExecute := bDriveDiagMessageAndNumber, Axis := RightTopLin.NcToPlc); // FB_SoEReadDiagNumber

// NETWORK 9
FB_SoEReadDiagNumber_LeftBottom(bExecute := bDriveDiagMessageAndNumber, Axis := LeftBottomLin.NcToPlc); // FB_SoEReadDiagNumber

// NETWORK 10
FB_SoEReadDiagNumber_RightBottom(bExecute := bDriveDiagMessageAndNumber, Axis := RightBottomLin.NcToPlc); // FB_SoEReadDiagNumber

// NETWORK 11
FB_SoEReadDiagNumber_PhaseUpper(bExecute := bDriveDiagMessageAndNumber, Axis := PhaseUpperLin.NcToPlc); // FB_SoEReadDiagNumber

// NETWORK 12
FB_SoEReadDiagNumber_PhaseLower(bExecute := bDriveDiagMessageAndNumber, Axis := PhaseLowerLin.NcToPlc); // FB_SoEReadDiagNumber

// NETWORK 13
FB_SoERead_GearNumerator_LeftTop(
    nIdn := P_0_IDN + 182,
    nElement := 16#40,
    pDstBuf := ADR(st_p182_LeftTop),
    cbBufLen := SIZEOF(st_p182_LeftTop),
    bExecute := bDriveDiagMessageAndNumber,
    Axis := LeftTopLin.NcToPlc); // FB_SoERead

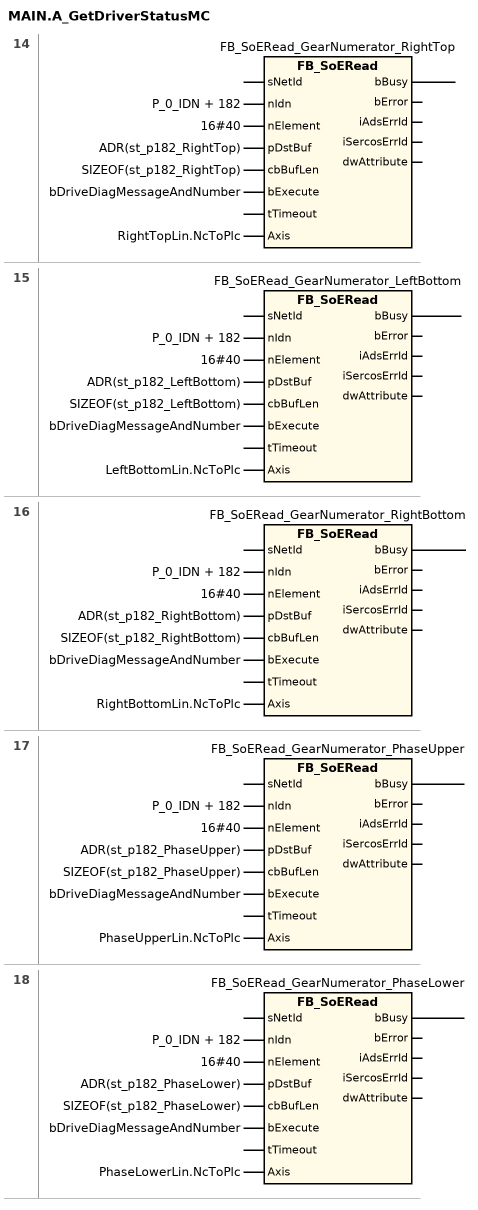
// NETWORK 14
FB_SoERead_GearNumerator_RightTop(
    nIdn := P_0_IDN + 182,
    nElement := 16#40,
    pDstBuf := ADR(st_p182_RightTop),
    cbBufLen := SIZEOF(st_p182_RightTop),
    bExecute := bDriveDiagMessageAndNumber,
    Axis := RightTopLin.NcToPlc); // FB_SoERead

// NETWORK 15
FB_SoERead_GearNumerator_LeftBottom(
    nIdn := P_0_IDN + 182,
    nElement := 16#40,
    pDstBuf := ADR(st_p182_LeftBottom),
    cbBufLen := SIZEOF(st_p182_LeftBottom),
    bExecute := bDriveDiagMessageAndNumber,
    Axis := LeftBottomLin.NcToPlc); // FB_SoERead

// NETWORK 16
FB_SoERead_GearNumerator_RightBottom(
    nIdn := P_0_IDN + 182,
    nElement := 16#40,
    pDstBuf := ADR(st_p182_RightBottom),
    cbBufLen := SIZEOF(st_p182_RightBottom),
    bExecute := bDriveDiagMessageAndNumber,
    Axis := RightBottomLin.NcToPlc); // FB_SoERead

// NETWORK 17
FB_SoERead_GearNumerator_PhaseUpper(
    nIdn := P_0_IDN + 182,
    nElement := 16#40,
    pDstBuf := ADR(st_p182_PhaseUpper),
    cbBufLen := SIZEOF(st_p182_PhaseUpper),
    bExecute := bDriveDiagMessageAndNumber,
    Axis := PhaseUpperLin.NcToPlc); // FB_SoERead

// NETWORK 18
FB_SoERead_GearNumerator_PhaseLower(
    nIdn := P_0_IDN + 182,
    nElement := 16#40,
    pDstBuf := ADR(st_p182_PhaseLower),
    cbBufLen := SIZEOF(st_p182_PhaseLower),
    bExecute := bDriveDiagMessageAndNumber,
    Axis := PhaseLowerLin.NcToPlc); // FB_SoERead

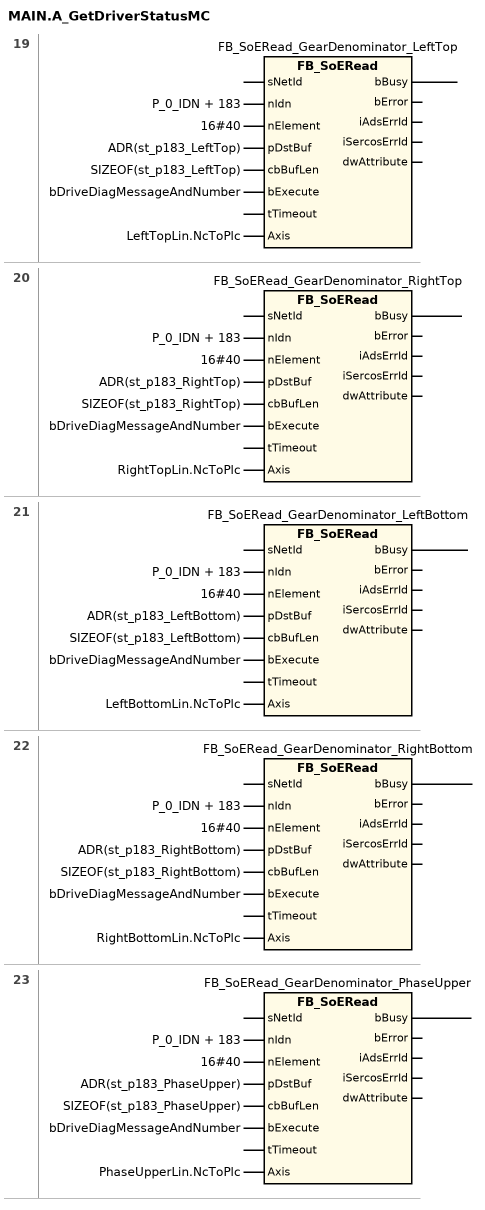
// NETWORK 19
FB_SoERead_GearDenominator_LeftTop(
    nIdn := P_0_IDN + 183,
    nElement := 16#40,
    pDstBuf := ADR(st_p183_LeftTop),
    cbBufLen := SIZEOF(st_p183_LeftTop),
    bExecute := bDriveDiagMessageAndNumber,
    Axis := LeftTopLin.NcToPlc); // FB_SoERead

// NETWORK 20
FB_SoERead_GearDenominator_RightTop(
    nIdn := P_0_IDN + 183,
    nElement := 16#40,
    pDstBuf := ADR(st_p183_RightTop),
    cbBufLen := SIZEOF(st_p183_RightTop),
    bExecute := bDriveDiagMessageAndNumber,
    Axis := RightTopLin.NcToPlc); // FB_SoERead

// NETWORK 21
FB_SoERead_GearDenominator_LeftBottom(
    nIdn := P_0_IDN + 183,
    nElement := 16#40,
    pDstBuf := ADR(st_p183_LeftBottom),
    cbBufLen := SIZEOF(st_p183_LeftBottom),
    bExecute := bDriveDiagMessageAndNumber,
    Axis := LeftBottomLin.NcToPlc); // FB_SoERead

// NETWORK 22
FB_SoERead_GearDenominator_RightBottom(
    nIdn := P_0_IDN + 183,
    nElement := 16#40,
    pDstBuf := ADR(st_p183_RightBottom),
    cbBufLen := SIZEOF(st_p183_RightBottom),
    bExecute := bDriveDiagMessageAndNumber,
    Axis := RightBottomLin.NcToPlc); // FB_SoERead

// NETWORK 23
FB_SoERead_GearDenominator_PhaseUpper(
    nIdn := P_0_IDN + 183,
    nElement := 16#40,
    pDstBuf := ADR(st_p183_PhaseUpper),
    cbBufLen := SIZEOF(st_p183_PhaseUpper),
    bExecute := bDriveDiagMessageAndNumber,
    Axis := PhaseUpperLin.NcToPlc); // FB_SoERead

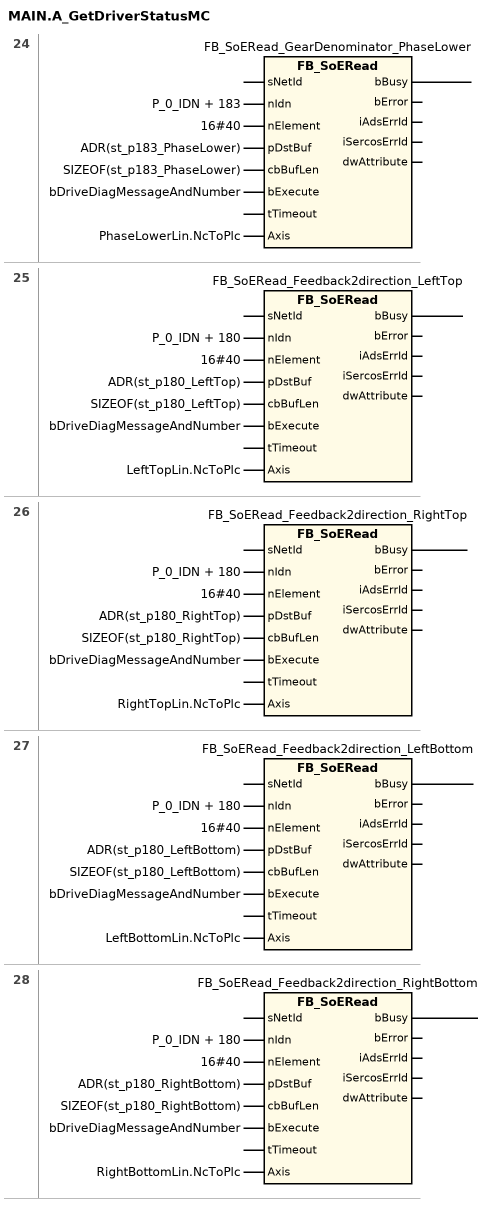
// NETWORK 24
FB_SoERead_GearDenominator_PhaseLower(
    nIdn := P_0_IDN + 183,
    nElement := 16#40,
    pDstBuf := ADR(st_p183_PhaseLower),
    cbBufLen := SIZEOF(st_p183_PhaseLower),
    bExecute := bDriveDiagMessageAndNumber,
    Axis := PhaseLowerLin.NcToPlc); // FB_SoERead

// NETWORK 25
FB_SoERead_Feedback2direction_LeftTop(
    nIdn := P_0_IDN + 180,
    nElement := 16#40,
    pDstBuf := ADR(st_p180_LeftTop),
    cbBufLen := SIZEOF(st_p180_LeftTop),
    bExecute := bDriveDiagMessageAndNumber,
    Axis := LeftTopLin.NcToPlc); // FB_SoERead

// NETWORK 26
FB_SoERead_Feedback2direction_RightTop(
    nIdn := P_0_IDN + 180,
    nElement := 16#40,
    pDstBuf := ADR(st_p180_RightTop),
    cbBufLen := SIZEOF(st_p180_RightTop),
    bExecute := bDriveDiagMessageAndNumber,
    Axis := RightTopLin.NcToPlc); // FB_SoERead

// NETWORK 27
FB_SoERead_Feedback2direction_LeftBottom(
    nIdn := P_0_IDN + 180,
    nElement := 16#40,
    pDstBuf := ADR(st_p180_LeftBottom),
    cbBufLen := SIZEOF(st_p180_LeftBottom),
    bExecute := bDriveDiagMessageAndNumber,
    Axis := LeftBottomLin.NcToPlc); // FB_SoERead

// NETWORK 28
FB_SoERead_Feedback2direction_RightBottom(
    nIdn := P_0_IDN + 180,
    nElement := 16#40,
    pDstBuf := ADR(st_p180_RightBottom),
    cbBufLen := SIZEOF(st_p180_RightBottom),
    bExecute := bDriveDiagMessageAndNumber,
    Axis := RightBottomLin.NcToPlc); // FB_SoERead

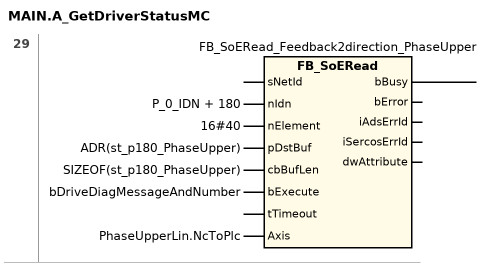
// NETWORK 29
FB_SoERead_Feedback2direction_PhaseUpper(
    nIdn := P_0_IDN + 180,
    nElement := 16#40,
    pDstBuf := ADR(st_p180_PhaseUpper),
    cbBufLen := SIZEOF(st_p180_PhaseUpper),
    bExecute := bDriveDiagMessageAndNumber,
    Axis := PhaseUpperLin.NcToPlc); // FB_SoERead
END_ACTION

ACTION A_GetMotorTemperature:
MotorTemperature_LeftTop:=UINT_TO_LREAL(MotorTemperature[0])/10;
MotorTemperature_RightTop:=UINT_TO_LREAL(MotorTemperature[1])/10;
MotorTemperature_LeftBottom:=UINT_TO_LREAL(MotorTemperature[2])/10;
MotorTemperature_RightBottom:=UINT_TO_LREAL(MotorTemperature[3])/10;
MotorTemperature_PhaseUpper:=UINT_TO_LREAL(MotorTemperature[4])/10;
MotorTemperature_PhaseLower:=UINT_TO_LREAL(MotorTemperature[5])/10;
END_ACTION

ACTION A_GetTemperatureSensorsData:
//sensor_1
dut_sensor_datas_1.data_byte[3]:=Sensor_Reading_1[0];
dut_sensor_datas_1.data_byte[2]:=Sensor_Reading_1[1];
dut_sensor_datas_1.data_byte[1]:=Sensor_Reading_1[2];
dut_sensor_datas_1.data_byte[0]:=Sensor_Reading_1[3];
TemperatureSensors_1:=DINT_TO_LREAL(LREAL_TO_DINT(dut_sensor_datas_1.data_lreal*100))/100;
//sensor_2
dut_sensor_datas_2.data_byte[3]:=Sensor_Reading_2[0];
dut_sensor_datas_2.data_byte[2]:=Sensor_Reading_2[1];
dut_sensor_datas_2.data_byte[1]:=Sensor_Reading_2[2];
dut_sensor_datas_2.data_byte[0]:=Sensor_Reading_2[3];
TemperatureSensors_2:=DINT_TO_LREAL(LREAL_TO_DINT(dut_sensor_datas_2.data_lreal*100))/100;
//sensor_3
dut_sensor_datas_3.data_byte[3]:=Sensor_Reading_3[0];
dut_sensor_datas_3.data_byte[2]:=Sensor_Reading_3[1];
dut_sensor_datas_3.data_byte[1]:=Sensor_Reading_3[2];
dut_sensor_datas_3.data_byte[0]:=Sensor_Reading_3[3];
TemperatureSensors_3:=DINT_TO_LREAL(LREAL_TO_DINT(dut_sensor_datas_3.data_lreal*100))/100;
//sensor_4
dut_sensor_datas_4.data_byte[3]:=Sensor_Reading_4[0];
dut_sensor_datas_4.data_byte[2]:=Sensor_Reading_4[1];
dut_sensor_datas_4.data_byte[1]:=Sensor_Reading_4[2];
dut_sensor_datas_4.data_byte[0]:=Sensor_Reading_4[3];
TemperatureSensors_4:=DINT_TO_LREAL(LREAL_TO_DINT(dut_sensor_datas_4.data_lreal*100))/100;
//sensor_5
dut_sensor_datas_5.data_byte[3]:=Sensor_Reading_5[0];
dut_sensor_datas_5.data_byte[2]:=Sensor_Reading_5[1];
dut_sensor_datas_5.data_byte[1]:=Sensor_Reading_5[2];
dut_sensor_datas_5.data_byte[0]:=Sensor_Reading_5[3];
TemperatureSensors_5:=DINT_TO_LREAL(LREAL_TO_DINT(dut_sensor_datas_5.data_lreal*100))/100;
//sensor_6
dut_sensor_datas_6.data_byte[3]:=Sensor_Reading_6[0];
dut_sensor_datas_6.data_byte[2]:=Sensor_Reading_6[1];
dut_sensor_datas_6.data_byte[1]:=Sensor_Reading_6[2];
dut_sensor_datas_6.data_byte[0]:=Sensor_Reading_6[3];
TemperatureSensors_6:=DINT_TO_LREAL(LREAL_TO_DINT(dut_sensor_datas_6.data_lreal*100))/100;
//sensor_7
dut_sensor_datas_7.data_byte[3]:=Sensor_Reading_7[0];
dut_sensor_datas_7.data_byte[2]:=Sensor_Reading_7[1];
dut_sensor_datas_7.data_byte[1]:=Sensor_Reading_7[2];
dut_sensor_datas_7.data_byte[0]:=Sensor_Reading_7[3];
TemperatureSensors_7:=DINT_TO_LREAL(LREAL_TO_DINT(dut_sensor_datas_7.data_lreal*100))/100;
//sensor_8
dut_sensor_datas_8.data_byte[3]:=Sensor_Reading_8[0];
dut_sensor_datas_8.data_byte[2]:=Sensor_Reading_8[1];
dut_sensor_datas_8.data_byte[1]:=Sensor_Reading_8[2];
dut_sensor_datas_8.data_byte[0]:=Sensor_Reading_8[3];
TemperatureSensors_8:=DINT_TO_LREAL(LREAL_TO_DINT(dut_sensor_datas_8.data_lreal*100))/100;
//计算temperature_gradient
temperature_gradient_2_To_1:=ABS(TemperatureSensors_2-TemperatureSensors_1);
temperature_gradient_3_To_2:=ABS(TemperatureSensors_3-TemperatureSensors_2);
temperature_gradient_5_To_4:=ABS(TemperatureSensors_5-TemperatureSensors_4);
temperature_gradient_6_To_5:=ABS(TemperatureSensors_6-TemperatureSensors_5);
temperature_gradient_max:=DINT_TO_LREAL(LREAL_TO_DINT(MAX(temperature_gradient_2_To_1,temperature_gradient_3_To_2,
							temperature_gradient_5_To_4,temperature_gradient_6_To_5)*100))/100;
//计算大梁上的温度平均值
temperature_average:=DINT_TO_LREAL(LREAL_TO_DINT((TemperatureSensors_1+TemperatureSensors_2+TemperatureSensors_3+TemperatureSensors_4
					+TemperatureSensors_5+TemperatureSensors_6)/6*100))/100;
					

//传感器温度状态：0：有传感器度数错误；1:常温；2:低温；3:常温和低温中间态
IF TemperatureSensors_1=0 OR TemperatureSensors_2=0 OR TemperatureSensors_3=0 
	OR TemperatureSensors_4=0 OR TemperatureSensors_5=0 OR TemperatureSensors_6=0 THEN	
	temperatureStatus:=0;//有传感器读数错误
ELSIF TemperatureSensors_1>=RoomTemperatureThreshold AND TemperatureSensors_2>=RoomTemperatureThreshold AND TemperatureSensors_3>=RoomTemperatureThreshold
	AND TemperatureSensors_4>=RoomTemperatureThreshold AND TemperatureSensors_5>=RoomTemperatureThreshold AND TemperatureSensors_6>=RoomTemperatureThreshold THEN	
	temperatureStatus:=1;//常温
ELSIF TemperatureSensors_1<=CryogenicTemperatureThreshold AND TemperatureSensors_1>77
	AND TemperatureSensors_2<=CryogenicTemperatureThreshold  AND TemperatureSensors_2>77
	AND TemperatureSensors_3<=CryogenicTemperatureThreshold  AND TemperatureSensors_3>77
	AND TemperatureSensors_4<=CryogenicTemperatureThreshold   AND TemperatureSensors_4>77
	AND TemperatureSensors_5<=CryogenicTemperatureThreshold  AND TemperatureSensors_5>77
	AND TemperatureSensors_6<=CryogenicTemperatureThreshold   AND TemperatureSensors_6>77 THEN	
	temperatureStatus:=2;//低温
ELSE
	temperatureStatus:=3;//常温和低温中间
END_IF
END_ACTION

ACTION A_InitAxisParameters:
(*ÖáÎ»ÖÃ¡¢ËÙ¶È¡¢PosDiff*)

	Pos_LeftTopLin:=DINT_TO_LREAL(LREAL_TO_DINT(LeftTopLin.NcToPlc.ActPos*100000))/100000;
	Pos_RightTopLin:=DINT_TO_LREAL(LREAL_TO_DINT(RightTopLin.NcToPlc.ActPos*100000))/100000;
	Pos_LeftBottomLin:=DINT_TO_LREAL(LREAL_TO_DINT(LeftBottomLin.NcToPlc.ActPos*100000))/100000;
	Pos_RightBottomLin:=DINT_TO_LREAL(LREAL_TO_DINT(RightBottomLin.NcToPlc.ActPos*100000))/100000;
	Pos_PhaseUpperLin:=DINT_TO_LREAL(LREAL_TO_DINT(PhaseUpperLin.NcToPlc.ActPos*100000))/100000;
	Pos_PhaseLowerLin:=DINT_TO_LREAL(LREAL_TO_DINT(PhaseLowerLin.NcToPlc.ActPos*100000))/100000;
	
	moveStatusLeftTop:=LeftTopLin.Status.Moving;
	moveStatusRightTop:=RightTopLin.Status.Moving;
	moveStatusLeftBottom:=LeftBottomLin.Status.Moving;
	moveStatusRightBottom:=RightBottomLin.Status.Moving;
	moveStatusPhaseUpper:=PhaseUpperLin.Status.Moving;
	moveStatusPhaseLower:=PhaseLowerLin.Status.Moving;
	
	moveStatusAllAxis:=moveStatusLeftTop AND moveStatusRightTop AND moveStatusLeftBottom AND moveStatusRightBottom;
	moveStatusAnyAxis:=moveStatusLeftTop OR moveStatusRightTop OR moveStatusLeftBottom OR moveStatusRightBottom;	
	Velo_LeftTopLin:=DINT_TO_LREAL(LREAL_TO_DINT(LeftTopLin.NcToPlc.ActVelo*100000))/100000;
	Velo_RightTopLin:=DINT_TO_LREAL(LREAL_TO_DINT(RightTopLin.NcToPlc.ActVelo*100000))/100000;
	Velo_LeftBottomLin:=DINT_TO_LREAL(LREAL_TO_DINT(LeftBottomLin.NcToPlc.ActVelo*100000))/100000;
	Velo_RightBottomLin:=DINT_TO_LREAL(LREAL_TO_DINT(RightBottomLin.NcToPlc.ActVelo*100000))/100000;
	Velo_PhaseUpperLin:=DINT_TO_LREAL(LREAL_TO_DINT(PhaseUpperLin.NcToPlc.ActVelo*100000))/100000;
	Velo_PhaseLowerLin:=DINT_TO_LREAL(LREAL_TO_DINT(PhaseLowerLin.NcToPlc.ActVelo*100000))/100000;
	
	PosDiff_LeftTopLin_actual:=DINT_TO_LREAL(LREAL_TO_DINT(LeftTopLin.NcToPlc.PosDiff*100000))/100000;
	PosDiff_RightTopLin_actual:=DINT_TO_LREAL(LREAL_TO_DINT(RightTopLin.NcToPlc.PosDiff*100000))/100000;
	PosDiff_LeftBottomLin_actual:=DINT_TO_LREAL(LREAL_TO_DINT(LeftBottomLin.NcToPlc.PosDiff*100000))/100000;
	PosDiff_RightBottomLin_actual:=DINT_TO_LREAL(LREAL_TO_DINT(RightBottomLin.NcToPlc.PosDiff*100000))/100000;
	PosDiff_PhaseUpperLin_actual:=DINT_TO_LREAL(LREAL_TO_DINT(PhaseUpperLin.NcToPlc.PosDiff*100000))/100000;
	PosDiff_PhaseLowerLin_actual:=DINT_TO_LREAL(LREAL_TO_DINT(PhaseLowerLin.NcToPlc.PosDiff*100000))/100000;;

	//Torque
	Torque_LeftTopLin:=LeftTopLin.NcToPlc.ActTorque;
	Torque_RightTopLin:=RightTopLin.NcToPlc.ActTorque;
	Torque_LeftBottomLin:=LeftBottomLin.NcToPlc.ActTorque;
	Torque_RightBottomLin:=RightBottomLin.NcToPlc.ActTorque;
	Torque_PhaseUpperLin:=LeftBottomLin.NcToPlc.ActTorque;
	Torque_PhaseLowerLin:=RightBottomLin.NcToPlc.ActTorque;
	
	LeftTopLin.ReadStatus();
	RightTopLin.ReadStatus();
	LeftBottomLin.ReadStatus();
	RightBottomLin.ReadStatus();
	PhaseUpperLin.ReadStatus();
	PhaseLowerLin.ReadStatus();

(*Motor Pos Velo Lagdistance status get*)
	//Position
	Pos_LeftTopMotor:=DINT_TO_LREAL(LREAL_TO_DINT(LeftTopMotor.NcToPlc.ActPos*100000))/100000;
	Pos_RightTopMotor:=DINT_TO_LREAL(LREAL_TO_DINT(RightTopMotor.NcToPlc.ActPos*100000))/100000;
	Pos_LeftBottomMotor:=DINT_TO_LREAL(LREAL_TO_DINT(LeftBottomMotor.NcToPlc.ActPos*100000))/100000;
	Pos_RightBottomMotor:=DINT_TO_LREAL(LREAL_TO_DINT(RightBottomMotor.NcToPlc.ActPos*100000))/100000;
	Pos_PhaseUpperMotor:=DINT_TO_LREAL(LREAL_TO_DINT(PhaseUpperMotor.NcToPlc.ActPos*100000))/100000;
	Pos_PhaseLowerMotor:=DINT_TO_LREAL(LREAL_TO_DINT(PhaseLowerMotor.NcToPlc.ActPos*100000))/100000;
	//Moving status
	moveStatusLeftTopMotor:=LeftTopMotor.Status.Moving;
	moveStatusRightTopMotor:=RightTopMotor.Status.Moving;
	moveStatusLeftBottomMotor:=LeftBottomMotor.Status.Moving;
	moveStatusRightBottomMotor:=RightBottomMotor.Status.Moving;
	moveStatusPhaseUpperMotor:=PhaseUpperMotor.Status.Moving;
	moveStatusPhaseLowerMotor:=PhaseLowerMotor.Status.Moving;
	moveStatusAllAxisMotor:=moveStatusLeftTopMotor AND moveStatusRightTopMotor AND moveStatusLeftBottomMotor AND moveStatusRightBottomMotor;
	moveStatusAnyAxisMotor:=moveStatusLeftTopMotor OR moveStatusRightTopMotor OR moveStatusLeftBottomMotor OR moveStatusRightBottomMotor;
	//Velocity
	Velo_LeftTopMotor:=DINT_TO_LREAL(LREAL_TO_DINT(LeftTopMotor.NcToPlc.ActVelo*100000))/100000;
	Velo_RightTopMotor:=DINT_TO_LREAL(LREAL_TO_DINT(RightTopMotor.NcToPlc.ActVelo*100000))/100000;
	Velo_LeftBottomMotor:=DINT_TO_LREAL(LREAL_TO_DINT(LeftBottomMotor.NcToPlc.ActVelo*100000))/100000;
	Velo_RightBottomMotor:=DINT_TO_LREAL(LREAL_TO_DINT(RightBottomMotor.NcToPlc.ActVelo*100000))/100000;
	Velo_PhaseUpperMotor:=DINT_TO_LREAL(LREAL_TO_DINT(PhaseUpperMotor.NcToPlc.ActVelo*100000))/100000;
	Velo_PhaseLowerMotor:=DINT_TO_LREAL(LREAL_TO_DINT(PhaseLowerMotor.NcToPlc.ActVelo*100000))/100000;
	//LagDistance
	PosDiff_LeftTopMotor_actual:=DINT_TO_LREAL(LREAL_TO_DINT(LeftTopMotor.NcToPlc.PosDiff*100000))/100000;
	PosDiff_RightTopMotor_actual:=DINT_TO_LREAL(LREAL_TO_DINT(RightTopMotor.NcToPlc.PosDiff*100000))/100000;
	PosDiff_LeftBottomMotor_actual:=DINT_TO_LREAL(LREAL_TO_DINT(LeftBottomMotor.NcToPlc.PosDiff*100000))/100000;
	PosDiff_RightBottomMotor_actual:=DINT_TO_LREAL(LREAL_TO_DINT(RightBottomMotor.NcToPlc.PosDiff*100000))/100000;
	PosDiff_PhaseUpperMotor_actual:=DINT_TO_LREAL(LREAL_TO_DINT(PhaseUpperMotor.NcToPlc.PosDiff*100000))/100000;
	PosDiff_PhaseLowerMotor_actual:=DINT_TO_LREAL(LREAL_TO_DINT(PhaseLowerMotor.NcToPlc.PosDiff*100000))/100000;
	//Torque
	Torque_LeftTopMotor:=LeftTopMotor.NcToPlc.ActTorque;
	Torque_RightTopMotor:=RightTopMotor.NcToPlc.ActTorque;
	Torque_LeftBottomMotor:=LeftBottomMotor.NcToPlc.ActTorque;
	Torque_RightBottomMotor:=RightBottomMotor.NcToPlc.ActTorque;
	Torque_PhaseUpperMotor:=PhaseUpperMotor.NcToPlc.ActTorque;
	Torque_PhaseLowerMotor:=PhaseLowerMotor.NcToPlc.ActTorque;

	LeftTopMotor.ReadStatus();
	RightTopMotor.ReadStatus();
	LeftBottomMotor.ReadStatus();
	RightBottomMotor.ReadStatus();
	PhaseUpperMotor.ReadStatus();
	PhaseLowerMotor.ReadStatus();
	//
	//get Delta
	//
	//Delta Pos
	DeltaPos_LeftTop:=Pos_LeftTopLin - Pos_LeftTopMotor;
	DeltaPos_RightTop:=Pos_RightTopLin - Pos_RightTopMotor;
	DeltaPos_LeftBottom:=Pos_LeftBottomLin - Pos_LeftBottomMotor;
	DeltaPos_RightBottom:=Pos_RightBottomLin - Pos_RightBottomMotor;
	DeltaPos_PhaseUpper:=Pos_PhaseUpperLin - Pos_PhaseUpperMotor;
	DeltaPos_PhaseLower:=Pos_PhaseLowerLin - Pos_PhaseLowerMotor;
	//Delta Velocity	
	DeltaVelo_LeftTop:=Velo_LeftTopLin - Velo_LeftTopMotor;
	DeltaVelo_RightTop:=Velo_RightTopLin - Velo_RightTopMotor;
	DeltaVelo_LeftBottom:=Velo_LeftBottomLin - Velo_LeftBottomMotor;
	DeltaVelo_RightBottom:=Velo_RightBottomLin - Velo_RightBottomMotor;
	DeltaVelo_PhaseUpper:=Velo_PhaseUpperLin - Velo_PhaseUpperMotor;
	DeltaVelo_PhaseLower:=Velo_PhaseLowerLin - Velo_PhaseLowerMotor;
	//Delta lagDistance
	DeltaPosDiff_LeftTop_actual:=PosDiff_LeftTopLin_actual - PosDiff_LeftTopMotor_actual;
	DeltaPosDiff_RightTop_actual:=PosDiff_RightTopLin_actual - PosDiff_RightTopMotor_actual;
	DeltaPosDiff_LeftBottom_actual:=PosDiff_LeftBottomLin_actual - PosDiff_LeftBottomMotor_actual;
	DeltaPosDiff_RightBottom_actual:=PosDiff_RightBottomLin_actual - PosDiff_RightBottomMotor_actual;	
	DeltaPosDiff_PhaseUpper_actual:=PosDiff_PhaseUpperLin_actual - PosDiff_PhaseUpperMotor_actual;
	DeltaPosDiff_PhaseLower_actual:=PosDiff_PhaseLowerLin_actual - PosDiff_PhaseLowerMotor_actual;	
	//Delta Torque
	DeltaTorque_LeftTop:=Torque_LeftTopLin - Torque_LeftTopMotor;
	DeltaTorque_RightTop:=Torque_RightTopLin - Torque_RightTopMotor;
	DeltaTorque_LeftBottom:=Torque_LeftBottomLin -Torque_LeftBottomMotor;
	DeltaTorque_RightBottom:=Torque_RightBottomLin - Torque_RightBottomMotor;
	DeltaTorque_PhaseUpper:=Torque_PhaseUpperLin -Torque_PhaseUpperMotor;
	DeltaTorque_PhaseLower:=Torque_PhaseLowerLin - Torque_PhaseLowerMotor;
END_ACTION

ACTION A_InitRecipeParameters:
CASE state_loadParameters OF
	0:
		LoadParameter:=TRUE;
		Read_R_TRIG(CLK:=LoadParameter , Q=> );
		IF Read_R_TRIG.Q THEN
			state_loadParameters:=1;
		END_IF
	1:
		 ReturnDwordLoad:=RecipeManCommands.LoadAndWriteRecipe(RecipeDefinitionName:='Recipes' , RecipeName:='ParametersAK');
    	 LoadParameter:=FALSE;
		 IF ReturnDwordLoad<>0 THEN
		 	state_loadParameters:=-100;
		ELSE
			LoadRecipeParameters:=TRUE;
			LoadParameter:=FALSE;
			state_loadParameters:=88;
	 	END_IF
	88:
		loadParametersDone:=TRUE;
	-100:
		loadParametersDone:=FALSE;
		Error:=TRUE;
		ErrorId:=101;
		ErrorDescription:='LoadRecipeParameters Error';
		Plc_EmergencyStop:=FALSE;
END_CASE

////Save_R_TRIG(CLK:=SaveParameter , Q=> );
//Read_R_TRIG(CLK:=LoadParameter , Q=> );
//IF Save_R_TRIG.Q THEN  //将plc数据以文件形式保存在工控机中
//	 RecipeManCommands.CreateRecipe(RecipeDefinitionName:='Recipes' , RecipeName:='Parameters' );
//	 RecipeManCommands.ReadAndSaveRecipe(RecipeDefinitionName:='Recipes' , RecipeName:='Parameters' );
//	 SaveParameter:=FALSE;
//END_IF
//IF Read_R_TRIG.Q THEN  //将工控机中的文件数据读取到plc中
//     ReturnDwordLoad:=RecipeManCommands.LoadAndWriteRecipe(RecipeDefinitionName:='Recipes' , RecipeName:='Parameters');
//     LoadParameter:=FALSE;
//	 IF ReturnDwordLoad<>0 THEN
//		 Error:=TRUE;
//		 ErrorId:=101;
//		 ErrorDescription:='LoadRecipeParameters Error';
//		 Plc_EmergencyStop:=FALSE;
//	 END_IF
//END_IF
END_ACTION

ACTION A_KillOpcIocShellExe:
R_TRIG_Exekill(CLK:=bExe_Kill_Prog, Q=> );
CASE Exe_kill_step OF
	0:
		IF R_TRIG_Exekill.Q THEN
			NT_StartProcess_Kill.START:=FALSE;
			NT_StartProcess_Kill.PATHSTR:='C:\HZB\OpcIocShell\IDControlIOC\killcmd.bat';
			//NT_StartProcess_Kill.DIRNAME:='C:\Program Files (x86)\HZB\OpcIocShell\bin\opcIocShell.exe';
			Exe_kill_step:=10;
		END_IF;
	10:
		NT_StartProcess_Kill.START:=TRUE;
		Exe_kill_step:=20;
	20:
		IF NT_StartProcess_Kill.ERR THEN
			Exe_kill_step:=0;
		ELSE
			Exe_kill_step:=30;
		END_IF;

	30:
		NT_StartProcess_Kill.START:=TRUE;
		Exe_kill_step:=40;
	40:
		IF NOT NT_StartProcess_Kill.BUSY THEN
			NT_StartProcess_Kill.START:=FALSE;
			Exe_Kill_Done:=TRUE;
			Exe_kill_step:=0;
		END_IF;
END_CASE;

NT_StartProcess_Kill(
	NETID:='' ,
	PATHSTR:= ,
	DIRNAME:= , 
	COMNDLINE:= , 
	START:= ,
	ERRID=> );
END_ACTION

ACTION A_LEHeartBeatMonitor:
//monitor only while power on and not simulation or not use LE
IF NOT st_Power THEN
	RETURN;
END_IF
(**)
IF simulation THEN
	RETURN;
END_IF
IF NOT USELinearEncoder THEN
	RETURN;
END_IF

// 初始化
IF LEHeartBeatFirstScan THEN
    Velo_LeftTopLin_Last := LeftTopLin.NcToPlc.ActVelo;
    Velo_RightTopLin_Last := RightTopLin.NcToPlc.ActVelo;
    Velo_LeftBottomLin_Last := LeftBottomLin.NcToPlc.ActVelo;
    Velo_RightBottomLin_Last := RightBottomLin.NcToPlc.ActVelo;
    Velo_PhaseUpperLin_Last := PhaseUpperLin.NcToPlc.ActVelo;
    Velo_PhaseLowerLin_Last := PhaseLowerLin.NcToPlc.ActVelo;
    LEHeartBeatFirstScan := FALSE;
END_IF;

// 计算光栅前后速度差，速度差比位置差更敏感
DeltaVelo_LeftTopLin := ABS(LeftTopLin.NcToPlc.ActVelo - Velo_LeftTopLin_Last);
DeltaVelo_RightTopLin := ABS(RightTopLin.NcToPlc.ActVelo - Velo_RightTopLin_Last);
DeltaVelo_LeftBottomLin := ABS(LeftBottomLin.NcToPlc.ActVelo - Velo_LeftBottomLin_Last);
DeltaVelo_RightBottomLin := ABS(RightBottomLin.NcToPlc.ActVelo - Velo_RightBottomLin_Last);
DeltaVelo_PhaseUpperLin := ABS(PhaseUpperLin.NcToPlc.ActVelo - Velo_PhaseUpperLin_Last);
DeltaVelo_PhaseLowerLin := ABS(PhaseLowerLin.NcToPlc.ActVelo - Velo_PhaseLowerLin_Last);
//LeftTop monitor
IF DeltaVelo_LeftTopLin > LEHeartBeatDeadZone THEN
    // 有变动，光栅正常，计数器归零，更新位置,重置所有状态
    StableTimer_LeftTopLin(IN := FALSE, PT := LEHeartBeatAlarmTime);
    Alarm_LeftTopLin := FALSE;
    Velo_LeftTopLin_Last := LeftTopLin.NcToPlc.ActVelo;  // 
    StableTime_LeftTopLin := T#0S;
	IsInitialPositionSet_LeftTop:=FALSE;
	Alarm_LeftTopMotorPos:=FALSE;
	Alarm_LeftTopMotorVelo:=FALSE;
ELSE
    //一点变动没有了，光栅异常，开始计时
    StableTimer_LeftTopLin(
        IN := TRUE,
        PT := LEHeartBeatAlarmTime,
        ET => StableTime_LeftTopLin
    );
	//记录电机初始位置，后后续对比做准备
	IF NOT IsInitialPositionSet_LeftTop THEN
        Pos_LeftTopMotor_Initial := Pos_LeftTopMotor;  // 记录初始位置
        IsInitialPositionSet_LeftTop := TRUE;
   	END_IF;
    
    // 100ms速度完全不变，开始监控电机速度和位置
    IF StableTimer_LeftTopLin.Q THEN
        Alarm_LeftTopLin := TRUE;  // 
			//电机位置对比及监测
			MotorPosChange_LeftTop:=ABS( Pos_LeftTopMotor-Pos_LeftTopMotor_Initial);
			IF MotorPosChange_LeftTop > Threshold_LeftTopMotorPos THEN
				Alarm_LeftTopMotorPos:=TRUE;
				ErrorID:=5001;
				ErrorDescription:='5001';
				Error:=TRUE;
				FB_PlcEmergencyStop();
				LED_Error:=TRUE;
			ELSE
				Alarm_LeftTopMotorPos:=FALSE;
			END_IF
			//电机速度监测
			IF Velo_LeftTopMotor > Threshold_LeftTopMotorVelo THEN
				Alarm_LeftTopMotorVelo:=TRUE;
				ErrorID:=5002;
				ErrorDescription:='5002';
				Error:=TRUE;
				FB_PlcEmergencyStop();
				LED_Error:=TRUE;
			ELSE
				Alarm_LeftTopMotorVelo:=FALSE;
			END_IF
    ELSE
        Alarm_LeftTopLin := FALSE;
	END_IF
END_IF
//RightTop monitor
IF DeltaVelo_RightTopLin > LEHeartBeatDeadZone THEN
    // 有变动，光栅正常，计数器归零，更新位置,重置所有状态
    StableTimer_RightTopLin(IN := FALSE, PT := LEHeartBeatAlarmTime);
    Alarm_RightTopLin := FALSE;
    Velo_RightTopLin_Last := RightTopLin.NcToPlc.ActVelo;  // 
    StableTime_RightTopLin := T#0S;
	IsInitialPositionSet_RightTop:=FALSE;
	Alarm_RightTopMotorPos:=FALSE;
	Alarm_RightTopMotorVelo:=FALSE;
ELSE
    //一点变动没有了，光栅异常，开始计时
    StableTimer_RightTopLin(
        IN := TRUE,
        PT :=LEHeartBeatAlarmTime,
        ET => StableTime_RightTopLin
    );
	//记录电机初始位置，后后续对比做准备
	IF NOT IsInitialPositionSet_RightTop THEN
        Pos_RightTopMotor_Initial := Pos_RightTopMotor;  // 记录初始位置
        IsInitialPositionSet_RightTop := TRUE;
   	END_IF;
    
    // 100ms速度完全不变，开始监控电机速度和位置
    IF StableTimer_RightTopLin.Q THEN
        Alarm_RightTopLin := TRUE;  // 
			//电机位置对比及监测
			MotorPosChange_RightTop:=ABS( Pos_RightTopMotor-Pos_RightTopMotor_Initial);
			IF MotorPosChange_RightTop > Threshold_RightTopMotorPos THEN
				Alarm_RightTopMotorPos:=TRUE;
				ErrorID:=5003;
				ErrorDescription:='5003';
				Error:=TRUE;
				FB_PlcEmergencyStop();
				LED_Error:=TRUE;
			ELSE
				Alarm_RightTopMotorPos:=FALSE;
			END_IF
			//电机速度监测
			IF Velo_RightTopMotor > Threshold_RightTopMotorVelo THEN
				Alarm_RightTopMotorVelo:=TRUE;
				ErrorID:=5004;
				ErrorDescription:='5004';
				Error:=TRUE;
				FB_PlcEmergencyStop();
				LED_Error:=TRUE;
			ELSE
				Alarm_RightTopMotorVelo:=FALSE;
			END_IF
    ELSE
        Alarm_RightTopLin := FALSE;
	END_IF
END_IF
//LeftBottom monitor
IF DeltaVelo_LeftBottomLin > LEHeartBeatDeadZone THEN
    // 有变动，光栅正常，计数器归零，更新位置,重置所有状态
    StableTimer_LeftBottomLin(IN := FALSE, PT := LEHeartBeatAlarmTime);
    Alarm_LeftBottomLin := FALSE;
    Velo_LeftBottomLin_Last := LeftBottomLin.NcToPlc.ActVelo;  // 
    StableTime_LeftBottomLin := T#0S;
	IsInitialPositionSet_LeftBottom:=FALSE;
	Alarm_LeftBottomMotorPos:=FALSE;
	Alarm_LeftBottomMotorVelo:=FALSE;
ELSE
    //一点变动没有了，光栅异常，开始计时
    StableTimer_LeftBottomLin(
        IN := TRUE,
        PT := LEHeartBeatAlarmTime,
        ET => StableTime_LeftBottomLin
    );
	//记录电机初始位置，后后续对比做准备
	IF NOT IsInitialPositionSet_LeftBottom THEN
        Pos_LeftBottomMotor_Initial := Pos_LeftBottomMotor;  // 记录初始位置
        IsInitialPositionSet_LeftBottom := TRUE;
   	END_IF;
    
    // 100ms速度完全不变，开始监控电机速度和位置
    IF StableTimer_LeftBottomLin.Q THEN
        Alarm_LeftBottomLin := TRUE;  // 
			//电机位置对比及监测
			MotorPosChange_LeftBottom:=ABS( Pos_LeftBottomMotor-Pos_LeftBottomMotor_Initial);
			IF MotorPosChange_LeftBottom > Threshold_LeftBottomMotorPos THEN
				Alarm_LeftBottomMotorPos:=TRUE;
				ErrorID:=5005;
				ErrorDescription:='5005';
				Error:=TRUE;
				FB_PlcEmergencyStop();
				LED_Error:=TRUE;
			ELSE
				Alarm_LeftBottomMotorPos:=FALSE;
			END_IF
			//电机速度监测
			IF Velo_LeftBottomMotor > Threshold_LeftBottomMotorVelo THEN
				Alarm_LeftBottomMotorVelo:=TRUE;
				ErrorID:=5006;
				ErrorDescription:='5006';
				Error:=TRUE;
				FB_PlcEmergencyStop();
				LED_Error:=TRUE;
			ELSE
				Alarm_LeftBottomMotorVelo:=FALSE;
			END_IF
    ELSE
        Alarm_LeftBottomLin := FALSE;
	END_IF
END_IF
//RightBottom monitor
IF DeltaVelo_RightBottomLin > LEHeartBeatDeadZone THEN
    // 有变动，光栅正常，计数器归零，更新位置,重置所有状态
    StableTimer_RightBottomLin(IN := FALSE, PT := LEHeartBeatAlarmTime);
    Alarm_RightBottomLin := FALSE;
    Velo_RightBottomLin_Last := RightBottomLin.NcToPlc.ActVelo;  // 
    StableTime_RightBottomLin := T#0S;
	IsInitialPositionSet_RightBottom:=FALSE;
	Alarm_RightBottomMotorPos:=FALSE;
	Alarm_RightBottomMotorVelo:=FALSE;
ELSE
    //一点变动没有了，光栅异常，开始计时
    StableTimer_RightBottomLin(
        IN := TRUE,
        PT := LEHeartBeatAlarmTime,
        ET => StableTime_RightBottomLin
    );
	//记录电机初始位置，后后续对比做准备
	IF NOT IsInitialPositionSet_RightBottom THEN
        Pos_RightBottomMotor_Initial := Pos_RightBottomMotor;  // 记录初始位置
        IsInitialPositionSet_RightBottom := TRUE;
   	END_IF;
    
    // 100ms速度完全不变，开始监控电机速度和位置
    IF StableTimer_RightBottomLin.Q THEN
        Alarm_RightBottomLin := TRUE;  // 
			//电机位置对比及监测
			MotorPosChange_RightBottom:=ABS( Pos_RightBottomMotor-Pos_RightBottomMotor_Initial);
			IF MotorPosChange_RightBottom > Threshold_RightBottomMotorPos THEN
				Alarm_RightBottomMotorPos:=TRUE;
				ErrorID:=5007;
				ErrorDescription:='5007';
				Error:=TRUE;
				FB_PlcEmergencyStop();
				LED_Error:=TRUE;
			ELSE
				Alarm_RightBottomMotorPos:=FALSE;
			END_IF
			//电机速度监测
			IF Velo_RightBottomMotor > Threshold_RightBottomMotorVelo THEN
				Alarm_RightBottomMotorVelo:=TRUE;
				ErrorID:=5008;
				ErrorDescription:='5008';
				Error:=TRUE;
				FB_PlcEmergencyStop();
				LED_Error:=TRUE;
			ELSE
				Alarm_RightBottomMotorVelo:=FALSE;
			END_IF
    ELSE
        Alarm_RightBottomLin := FALSE;
	END_IF
END_IF
//PhaseUpper monitor
IF DeltaVelo_PhaseUpperLin > LEHeartBeatDeadZone THEN
    // 有变动，光栅正常，计数器归零，更新位置,重置所有状态
    StableTimer_PhaseUpperLin(IN := FALSE, PT := LEHeartBeatAlarmTime);
    Alarm_PhaseUpperLin := FALSE;
    Velo_PhaseUpperLin_Last := PhaseUpperLin.NcToPlc.ActVelo;  // 
    StableTime_PhaseUpperLin := T#0S;
	IsInitialPositionSet_PhaseUpper:=FALSE;
	Alarm_PhaseUpperMotorPos:=FALSE;
	Alarm_PhaseUpperMotorVelo:=FALSE;
ELSE
    //一点变动没有了，光栅异常，开始计时
    StableTimer_PhaseUpperLin(
        IN := TRUE,
        PT := LEHeartBeatAlarmTime,
        ET => StableTime_PhaseUpperLin
    );
	//记录电机初始位置，后后续对比做准备
	IF NOT IsInitialPositionSet_PhaseUpper THEN
        Pos_PhaseUpperMotor_Initial := Pos_PhaseUpperMotor;  // 记录初始位置
        IsInitialPositionSet_PhaseUpper := TRUE;
   	END_IF;
    
    // 100ms速度完全不变，开始监控电机速度和位置
    IF StableTimer_PhaseUpperLin.Q THEN
        Alarm_PhaseUpperLin := TRUE;  // 
			//电机位置对比及监测
			MotorPosChange_PhaseUpper:=ABS( Pos_PhaseUpperMotor-Pos_PhaseUpperMotor_Initial);
			IF MotorPosChange_PhaseUpper > Threshold_PhaseUpperMotorPos THEN
				Alarm_PhaseUpperMotorPos:=TRUE;
				ErrorID:=5009;
				ErrorDescription:='5009';
				Error:=TRUE;
				FB_PlcEmergencyStop();
				LED_Error:=TRUE;
			ELSE
				Alarm_PhaseUpperMotorPos:=FALSE;
			END_IF
			//电机速度监测
			IF Velo_PhaseUpperMotor > Threshold_PhaseUpperMotorVelo THEN
				Alarm_PhaseUpperMotorVelo:=TRUE;
				ErrorID:=5010;
				ErrorDescription:='5010';
				Error:=TRUE;
				FB_PlcEmergencyStop();
				LED_Error:=TRUE;
			ELSE
				Alarm_PhaseUpperMotorVelo:=FALSE;
			END_IF
    ELSE
        Alarm_PhaseUpperLin := FALSE;
	END_IF
END_IF
//PhaseLower monitor
IF DeltaVelo_PhaseLowerLin > LEHeartBeatDeadZone THEN
    // 有变动，光栅正常，计数器归零，更新位置,重置所有状态
    StableTimer_PhaseLowerLin(IN := FALSE, PT := LEHeartBeatAlarmTime);
    Alarm_PhaseLowerLin := FALSE;
    Velo_PhaseLowerLin_Last := PhaseLowerLin.NcToPlc.ActVelo;  // 
    StableTime_PhaseLowerLin := T#0S;
	IsInitialPositionSet_PhaseLower:=FALSE;
	Alarm_PhaseLowerMotorPos:=FALSE;
	Alarm_PhaseLowerMotorVelo:=FALSE;
ELSE
    //一点变动没有了，光栅异常，开始计时
    StableTimer_PhaseLowerLin(
        IN := TRUE,
        PT := LEHeartBeatAlarmTime,
        ET => StableTime_PhaseLowerLin
    );
	//记录电机初始位置，后后续对比做准备
	IF NOT IsInitialPositionSet_PhaseLower THEN
        Pos_PhaseLowerMotor_Initial := Pos_PhaseLowerMotor;  // 记录初始位置
        IsInitialPositionSet_PhaseLower := TRUE;
   	END_IF;
    
    // 100ms速度完全不变，开始监控电机速度和位置
    IF StableTimer_PhaseLowerLin.Q THEN
        Alarm_PhaseLowerLin := TRUE;  // 
			//电机位置对比及监测
			MotorPosChange_PhaseLower:=ABS( Pos_PhaseLowerMotor-Pos_PhaseLowerMotor_Initial);
			IF MotorPosChange_PhaseLower > Threshold_PhaseLowerMotorPos THEN
				Alarm_PhaseLowerMotorPos:=TRUE;
				ErrorID:=5011;
				ErrorDescription:='5011';
				Error:=TRUE;
				FB_PlcEmergencyStop();
				LED_Error:=TRUE;
			ELSE
				Alarm_PhaseLowerMotorPos:=FALSE;
			END_IF
			//电机速度监测
			IF Velo_PhaseLowerMotor > Threshold_PhaseLowerMotorVelo THEN
				Alarm_PhaseLowerMotorVelo:=TRUE;
				ErrorID:=5012;
				ErrorDescription:='5012';
				Error:=TRUE;
				FB_PlcEmergencyStop();
				LED_Error:=TRUE;
			ELSE
				Alarm_PhaseLowerMotorVelo:=FALSE;
			END_IF
    ELSE
        Alarm_PhaseLowerLin := FALSE;
	END_IF
END_IF
END_ACTION

ACTION A_LoadOpcIocShellExe:
R_TRIG_Exeload(CLK:=bExe_load_Prog, Q=> );
LoadOpcIocTON(PT:=T#10S);
CASE Exe_load_step OF
	0:
		LoadOpcIocTON.IN:=TRUE;
		IF R_TRIG_Exeload.Q THEN
			NT_StartProcess_Load.START:=FALSE;
			NT_StartProcess_Load.PATHSTR:='C:\HZB\OpcIocShell\IDControlIOC\startTwinCATOPCServer.bat';
			Exe_load_step:=10;
		END_IF;
	10:
		IF LoadOpcIocTON.Q THEN
			NT_StartProcess_Load.START:=TRUE;
			Exe_load_step:=20;
		END_IF
	20:
		LoadOpcIocTON.IN:=FALSE;
		IF NT_StartProcess_Load.ERR THEN
			Exe_load_step:=0;
		ELSE
			Exe_load_step:=30;
		END_IF;
	30:
		IF NOT NT_StartProcess_Load.BUSY THEN
			NT_StartProcess_Load.START:=FALSE;
			Exe_Load_Done:=TRUE;
			Exe_load_step:=0;
		END_IF;
END_CASE;

NT_StartProcess_Load(
	NETID:='' ,
	PATHSTR:= ,
	DIRNAME:= , 
	COMNDLINE:= , 
	START:= ,
	ERRID=> );
END_ACTION

